               //"PLC_LED_GREEN_1" := FALSE;
               //"PLC_LED_GREEN_2" := FALSE;
               //"PLC_LED_ORANGE_1" := TRUE;
               //"PLC_LED_ORANGE_2" := FALSE;
               //"PLC_LED_GREEN_CH" := FALSE;
               //"PLC_LED_RED_1" := FALSE;
               //"PLC_LED_RED_2" := TRUE;
               //"PLC_LED_RED_CH" := TRUE;

           4:  // Statement section case S5
               // GREEN = FALSE, YELLOW = FALSE, RED = TRUE
               // PED: RED = TRUE, GREEN = FALSE

               "DB_ProcessData".crossroad_output.trafficLightEast_green := FALSE;
               "DB_ProcessData".crossroad_output.trafficLightEast_red := TRUE;
               "DB_ProcessData".crossroad_output.trafficLightEast_yellow := FALSE;

               "DB_ProcessData".crossroad_output.trafficLightNorth_green := FALSE;
               "DB_ProcessData".crossroad_output.trafficLightNorth_red := TRUE;
               "DB_ProcessData".crossroad_output.trafficLightNorth_yellow := FALSE;

               "DB_ProcessData".crossroad_output.trafficLightSouth_green := FALSE;
               "DB_ProcessData".crossroad_output.trafficLightSouth_red := TRUE;
               "DB_ProcessData".crossroad_output.trafficLightSouth_yellow := FALSE;

               "DB_ProcessData".crossroad_output.trafficLightWest_green := FALSE;
               "DB_ProcessData".crossroad_output.trafficLightWest_red := TRUE;
               "DB_ProcessData".crossroad_output.trafficLightWest_yellow := FALSE;

               "DB_ProcessData".crossroad_output.pedestrianSouth1_green := FALSE;
               "DB_ProcessData".crossroad_output.pedestrianSouth1_red := TRUE;
               "DB_ProcessData".crossroad_output.pedestrianSouth2_green := FALSE;
               "DB_ProcessData".crossroad_output.pedestrianSouth2_red := TRUE;

               "DB_ProcessData".crossroad_output.pedestrianWest1_green := FALSE;
               "DB_ProcessData".crossroad_output.pedestrianWest1_red := TRUE;
               "DB_ProcessData".crossroad_output.pedestrianWest2_green := FALSE;
               "DB_ProcessData".crossroad_output.pedestrianWest2_red := TRUE;

               //"PLC_LED_GREEN_1" := FALSE;
               //"PLC_LED_GREEN_2" := FALSE;
               //"PLC_LED_ORANGE_1" := FALSE;
               //"PLC_LED_ORANGE_2" := FALSE;
               //"PLC_LED_GREEN_CH" := FALSE;
               //"PLC_LED_RED_1" := TRUE;
               //"PLC_LED_RED_2" := TRUE;
               //"PLC_LED_RED_CH" := TRUE;

           5:  // Statement section case S6
               // GREEN = FALSE, RED = TRUE, YELLOW = FALSE   // směr 1 (East, West)
               // GREEN = FALSE, RED = TRUE, YELLOW = TRUE    // směr 2 (North, South)
               // PED: RED = TRUE, GREEN = FALSE (pokud není Crossroad_Walk_EN)

               "DB_ProcessData".crossroad_output.trafficLightEast_green := FALSE;
               "DB_ProcessData".crossroad_output.trafficLightEast_red := TRUE;
               "DB_ProcessData".crossroad_output.trafficLightEast_yellow := FALSE;

               "DB_ProcessData".crossroad_output.trafficLightNorth_green := FALSE;
               "DB_ProcessData".crossroad_output.trafficLightNorth_red := TRUE;
               "DB_ProcessData".crossroad_output.trafficLightNorth_yellow := TRUE;

               "DB_ProcessData".crossroad_output.trafficLightSouth_green := FALSE;
               "DB_ProcessData".crossroad_output.trafficLightSouth_red := TRUE;
               "DB_ProcessData".crossroad_output.trafficLightSouth_yellow := TRUE;

               "DB_ProcessData".crossroad_output.trafficLightWest_green := FALSE;
               "DB_ProcessData".crossroad_output.trafficLightWest_red := TRUE;
               "DB_ProcessData".crossroad_output.trafficLightWest_yellow := FALSE;

               "DB_ProcessData".crossroad_output.pedestrianSouth1_green := FALSE;
               "DB_ProcessData".crossroad_output.pedestrianSouth1_red := TRUE;
               "DB_ProcessData".crossroad_output.pedestrianSouth2_green := FALSE;
               "DB_ProcessData".crossroad_output.pedestrianSouth2_red := TRUE;

               "DB_ProcessData".crossroad_output.pedestrianWest1_green := FALSE;
               "DB_ProcessData".crossroad_output.pedestrianWest1_red := TRUE;
               "DB_ProcessData".crossroad_output.pedestrianWest2_green := FALSE;
               "DB_ProcessData".crossroad_output.pedestrianWest2_red := TRUE;

               //"PLC_LED_GREEN_1" := FALSE;
               //"PLC_LED_GREEN_2" := FALSE;
               //"PLC_LED_ORANGE_1" := FALSE;
               //"PLC_LED_ORANGE_2" := TRUE;
               //"PLC_LED_GREEN_CH" := FALSE;
               //"PLC_LED_RED_1" := TRUE;
               //"PLC_LED_RED_2" := TRUE;

               //"PLC_LED_GREEN_CH" := FALSE;
               //"PLC_LED_RED_CH" := TRUE;

               IF "Crossroad_Walk_EN" THEN
                   "DB_ProcessData".crossroad_output.pedestrianSouth1_green := TRUE;
                   "DB_ProcessData".crossroad_output.pedestrianSouth1_red := FALSE;
                   "DB_ProcessData".crossroad_output.pedestrianSouth2_green := TRUE;
                   "DB_ProcessData".crossroad_output.pedestrianSouth2_red := FALSE;

                   "DB_ProcessData".crossroad_output.pedestrianWest1_green := TRUE;
                   "DB_ProcessData".crossroad_output.pedestrianWest1_red := FALSE;
                   "DB_ProcessData".crossroad_output.pedestrianWest2_green := TRUE;
                   "DB_ProcessData".crossroad_output.pedestrianWest2_red := FALSE;

                   //"PLC_LED_GREEN_CH" := TRUE;
                   //"PLC_LED_RED_CH" := FALSE;
               END_IF;

           6:  // Statement section case S7
               // GREEN = FALSE, RED = TRUE, YELLOW = FALSE   // směr 1 (East, West)
               // GREEN = TRUE, RED = FALSE, YELLOW = FALSE   // směr 2 (North, South)
               // PED: RED = TRUE, GREEN = FALSE (pokud není Crossroad_Walk_EN)

               "DB_ProcessData".crossroad_output.trafficLightEast_green := FALSE;
               "DB_ProcessData".crossroad_output.trafficLightEast_red := TRUE;
               "DB_ProcessData".crossroad_output.trafficLightEast_yellow := FALSE;

               "DB_ProcessData".crossroad_output.trafficLightNorth_green := TRUE;
               "DB_ProcessData".crossroad_output.trafficLightNorth_red := FALSE;
               "DB_ProcessData".crossroad_output.trafficLightNorth_yellow := FALSE;

               "DB_ProcessData".crossroad_output.trafficLightSouth_green := TRUE;
               "DB_ProcessData".crossroad_output.trafficLightSouth_red := FALSE;
               "DB_ProcessData".crossroad_output.trafficLightSouth_yellow := FALSE;

               "DB_ProcessData".crossroad_output.trafficLightWest_green := FALSE;
               "DB_ProcessData".crossroad_output.trafficLightWest_red := TRUE;
               "DB_ProcessData".crossroad_output.trafficLightWest_yellow := FALSE;

               "DB_ProcessData".crossroad_output.pedestrianSouth1_green := FALSE;
               "DB_ProcessData".crossroad_output.pedestrianSouth1_red := TRUE;
               "DB_ProcessData".crossroad_output.pedestrianSouth2_green := FALSE;
               "DB_ProcessData".crossroad_output.pedestrianSouth2_red := TRUE;

               "DB_ProcessData".crossroad_output.pedestrianWest1_green := FALSE;
               "DB_ProcessData".crossroad_output.pedestrianWest1_red := TRUE;
               "DB_ProcessData".crossroad_output.pedestrianWest2_green := FALSE;
               "DB_ProcessData".crossroad_output.pedestrianWest2_red := TRUE;

               //"PLC_LED_GREEN_1" := FALSE;
               //"PLC_LED_GREEN_2" := TRUE;
               //"PLC_LED_ORANGE_1" := FALSE;
               //"PLC_LED_ORANGE_2" := FALSE;
               //"PLC_LED_RED_1" := TRUE;
               //"PLC_LED_RED_2" := FALSE;

               //"PLC_LED_GREEN_CH" := FALSE;
               //"PLC_LED_RED_CH" := TRUE;

               IF "Crossroad_Walk_EN" THEN
                   "DB_ProcessData".crossroad_output.pedestrianSouth1_green := TRUE;
                   "DB_ProcessData".crossroad_output.pedestrianSouth1_red := FALSE;
                   "DB_ProcessData".crossroad_output.pedestrianSouth2_green := TRUE;
                   "DB_ProcessData".crossroad_output.pedestrianSouth2_red := FALSE;

                   "DB_ProcessData".crossroad_output.pedestrianWest1_green := TRUE;
                   "DB_ProcessData".crossroad_output.pedestrianWest1_red := FALSE;
                   "DB_ProcessData".crossroad_output.pedestrianWest2_green := TRUE;
                   "DB_ProcessData".crossroad_output.pedestrianWest2_red := FALSE;

                   //"PLC_LED_GREEN_CH" := TRUE;
                   //"PLC_LED_RED_CH" := FALSE;
               END_IF;

           7:  // Statement section case S8
               // GREEN = FALSE, RED = TRUE, YELLOW = FALSE   // směr 1 (East, West)
               // GREEN = FALSE, RED = FALSE, YELLOW = TRUE   // směr 2 (North, South)
               // PED: RED = TRUE, GREEN = FALSE

               "DB_ProcessData".crossroad_output.trafficLightEast_green := FALSE;
               "DB_ProcessData".crossroad_output.trafficLightEast_red := TRUE;
               "DB_ProcessData".crossroad_output.trafficLightEast_yellow := FALSE;

               "DB_ProcessData".crossroad_output.trafficLightNorth_green := FALSE;
               "DB_ProcessData".crossroad_output.trafficLightNorth_red := FALSE;
               "DB_ProcessData".crossroad_output.trafficLightNorth_yellow := TRUE;

               "DB_ProcessData".crossroad_output.trafficLightSouth_green := FALSE;
               "DB_ProcessData".crossroad_output.trafficLightSouth_red := FALSE;
               "DB_ProcessData".crossroad_output.trafficLightSouth_yellow := TRUE;

               "DB_ProcessData".crossroad_output.trafficLightWest_green := FALSE;
               "DB_ProcessData".crossroad_output.trafficLightWest_red := TRUE;
               "DB_ProcessData".crossroad_output.trafficLightWest_yellow := FALSE;

               "DB_ProcessData".crossroad_output.pedestrianSouth1_green := FALSE;
               "DB_ProcessData".crossroad_output.pedestrianSouth1_red := TRUE;
               "DB_ProcessData".crossroad_output.pedestrianSouth2_green := FALSE;
               "DB_ProcessData".crossroad_output.pedestrianSouth2_red := TRUE;

               "DB_ProcessData".crossroad_output.pedestrianWest1_green := FALSE;
               "DB_ProcessData".crossroad_output.pedestrianWest1_red := TRUE;
               "DB_ProcessData".crossroad_output.pedestrianWest2_green := FALSE;
               "DB_ProcessData".crossroad_output.pedestrianWest2_red := TRUE;

               //"PLC_LED_GREEN_1" := FALSE;
               //"PLC_LED_GREEN_2" := FALSE;
               //"PLC_LED_ORANGE_1" := FALSE;
               //"PLC_LED_ORANGE_2" := TRUE;
               //"PLC_LED_GREEN_CH" := FALSE;
               //"PLC_LED_RED_1" := TRUE;
               //"PLC_LED_RED_2" := FALSE;
               //"PLC_LED_RED_CH" := TRUE;

           8:  // Statement section case S9
               // GREEN = FALSE, YELLOW = FALSE, RED = TRUE
               // PED: RED = TRUE, GREEN = FALSE

               "DB_ProcessData".crossroad_output.trafficLightEast_green := FALSE;
               "DB_ProcessData".crossroad_output.trafficLightEast_red := TRUE;
               "DB_ProcessData".crossroad_output.trafficLightEast_yellow := FALSE;

               "DB_ProcessData".crossroad_output.trafficLightNorth_green := FALSE;
               "DB_ProcessData".crossroad_output.trafficLightNorth_red := TRUE;
               "DB_ProcessData".crossroad_output.trafficLightNorth_yellow := FALSE;

               "DB_ProcessData".crossroad_output.trafficLightSouth_green := FALSE;
               "DB_ProcessData".crossroad_output.trafficLightSouth_red := TRUE;
               "DB_ProcessData".crossroad_output.trafficLightSouth_yellow := FALSE;

               "DB_ProcessData".crossroad_output.trafficLightWest_green := FALSE;
               "DB_ProcessData".crossroad_output.trafficLightWest_red := TRUE;
               "DB_ProcessData".crossroad_output.trafficLightWest_yellow := FALSE;

               "DB_ProcessData".crossroad_output.pedestrianSouth1_green := FALSE;
               "DB_ProcessData".crossroad_output.pedestrianSouth1_red := TRUE;
               "DB_ProcessData".crossroad_output.pedestrianSouth2_green := FALSE;
               "DB_ProcessData".crossroad_output.pedestrianSouth2_red := TRUE;

               "DB_ProcessData".crossroad_output.pedestrianWest1_green := FALSE;
               "DB_ProcessData".crossroad_output.pedestrianWest1_red := TRUE;
               "DB_ProcessData".crossroad_output.pedestrianWest2_green := FALSE;
               "DB_ProcessData".crossroad_output.pedestrianWest2_red := TRUE;

               //"PLC_LED_GREEN_1" := FALSE;
               //"PLC_LED_GREEN_2" := FALSE;
               //"PLC_LED_ORANGE_1" := FALSE;
               //"PLC_LED_ORANGE_2" := FALSE;
               //"PLC_LED_GREEN_CH" := FALSE;
               //"PLC_LED_RED_1" := TRUE;
               //"PLC_LED_RED_2" := TRUE;
               //"PLC_LED_RED_CH" := TRUE;

               "Crossroad_Walk_EN" := FALSE;

           ELSE  // Statement section ELSE
               "DB_ProcessData".crossroad_output.trafficLightEast_green := FALSE;
               "DB_ProcessData".crossroad_output.trafficLightEast_red := FALSE;
               "DB_ProcessData".crossroad_output.trafficLightEast_yellow := FALSE;

               "DB_ProcessData".crossroad_output.trafficLightNorth_green := FALSE;
               "DB_ProcessData".crossroad_output.trafficLightNorth_red := FALSE;
               "DB_ProcessData".crossroad_output.trafficLightNorth_yellow := FALSE;

               "DB_ProcessData".crossroad_output.trafficLightSouth_green := FALSE;
               "DB_ProcessData".crossroad_output.trafficLightSouth_red := FALSE;
               "DB_ProcessData".crossroad_output.trafficLightSouth_yellow := FALSE;

               "DB_ProcessData".crossroad_output.trafficLightWest_green := FALSE;
               "DB_ProcessData".crossroad_output.trafficLightWest_red := FALSE;
               "DB_ProcessData".crossroad_output.trafficLightWest_yellow := FALSE;

               "DB_ProcessData".crossroad_output.pedestrianSouth1_green := FALSE;
               "DB_ProcessData".crossroad_output.pedestrianSouth1_red := FALSE;
               "DB_ProcessData".crossroad_output.pedestrianSouth2_green := FALSE;
               "DB_ProcessData".crossroad_output.pedestrianSouth2_red := FALSE;

               "DB_ProcessData".crossroad_output.pedestrianWest1_green := FALSE;
               "DB_ProcessData".crossroad_output.pedestrianWest1_red := FALSE;
               "DB_ProcessData".crossroad_output.pedestrianWest2_green := FALSE;
               "DB_ProcessData".crossroad_output.pedestrianWest2_red := FALSE;

               //"PLC_LED_GREEN_1" := FALSE;
               //"PLC_LED_GREEN_2" := FALSE;
               //"PLC_LED_ORANGE_1" := FALSE;
               //"PLC_LED_ORANGE_2" := FALSE;
               //"PLC_LED_RED_1" := FALSE;
               //"PLC_LED_RED_2" := FALSE;
               //"PLC_LED_GREEN_CH" := FALSE;
               //"PLC_LED_RED_CH" := FALSE;

               "Crossroad_Walk_EN" := FALSE;
       END_CASE;
   END_IF;
END_REGION

REGION Network 6 (SCL): Pedestrians bnts
   IF "DB_ProcessData".crossroad_input.btnSouthCrosswalk1 OR "DB_ProcessData".crossroad_input.btnSouthCrosswalk2 OR "DB_ProcessData".crossroad_input.btnWestCrosswalk1 OR "DB_ProcessData".crossroad_input.btnWestCrosswalk2 THEN
       "Crossroad_Walk_EN" := TRUE;
   END_IF;
END_REGION
END_FUNCTION

// folder: Crosswalk

FUNCTION "Crosswalk_MAIN" : Void   // FC1, LAD
{ S7_Optimized_Access := 'TRUE' }
VERSION : 0.1
BEGIN

REGION Network 1: Control
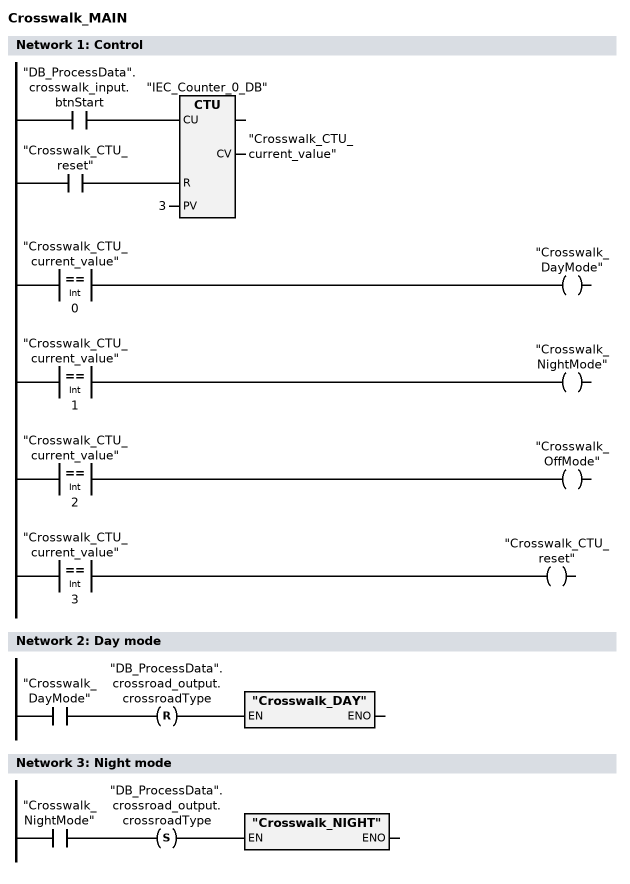
   "IEC_Counter_0_DB".CTU(CU := "DB_ProcessData".crosswalk_input.btnStart,
                          R := "Crosswalk_CTU_reset",
                          PV := 3,
                          CV => "Crosswalk_CTU_current_value");
   "Crosswalk_DayMode" := "Crosswalk_CTU_current_value" = 0;
   "Crosswalk_NightMode" := "Crosswalk_CTU_current_value" = 1;
   "Crosswalk_OffMode" := "Crosswalk_CTU_current_value" = 2;
   "Crosswalk_CTU_reset" := "Crosswalk_CTU_current_value" = 3;
END_REGION

REGION Network 2: Day mode
   RUNG wire#powerrail
      Contact( "Crosswalk_DayMode" )
      R_Coil( "DB_ProcessData".crossroad_output.crossroadType )
      "Crosswalk_DAY"()
   END_RUNG
   // the same network as SCL:
   IF "Crosswalk_DayMode" THEN
       "DB_ProcessData".crossroad_output.crossroadType := FALSE;
       "Crosswalk_DAY"();
   END_IF;
END_REGION

REGION Network 3: Night mode
   RUNG wire#powerrail
      Contact( "Crosswalk_NightMode" )
      S_Coil( "DB_ProcessData".crossroad_output.crossroadType )
      "Crosswalk_NIGHT"()
   END_RUNG
   // the same network as SCL:
   IF "Crosswalk_NightMode" THEN
       "DB_ProcessData".crossroad_output.crossroadType := TRUE;
       "Crosswalk_NIGHT"();
   END_IF;
END_REGION

REGION Network 4 (SCL): Off mode
   IF "Crosswalk_OffMode" = TRUE THEN
       "DB_ProcessData".crosswalk_output.pedestrianLightGreen1 := FALSE;
       "DB_ProcessData".crosswalk_output.pedestrianLightGreen2 := FALSE;
       "DB_ProcessData".crosswalk_output.pedestrianLightRed1 := FALSE;
       "DB_ProcessData".crosswalk_output.pedestrianLightRed2 := FALSE;
       "DB_ProcessData".crosswalk_output.trafficLightGreen1 := FALSE;
       "DB_ProcessData".crosswalk_output.trafficLightGreen2 := FALSE;
       "DB_ProcessData".crosswalk_output.trafficLightsRed1 := FALSE;
       "DB_ProcessData".crosswalk_output.trafficLightsRed2 := FALSE;
       "DB_ProcessData".crosswalk_output.trafficLightsYellow1 := FALSE;
       "DB_ProcessData".crosswalk_output.trafficLightsYellow2 := FALSE;
   END_IF;
END_REGION
END_FUNCTION

FUNCTION "Crosswalk_DAY" : Void   // FC2, LAD
{ S7_Optimized_Access := 'TRUE' }
VERSION : 0.1
   VAR_TEMP   // added for the SCL form of the ladder/FBD networks
      _w1 : Bool;
   END_VAR
BEGIN

REGION Network 1: Green
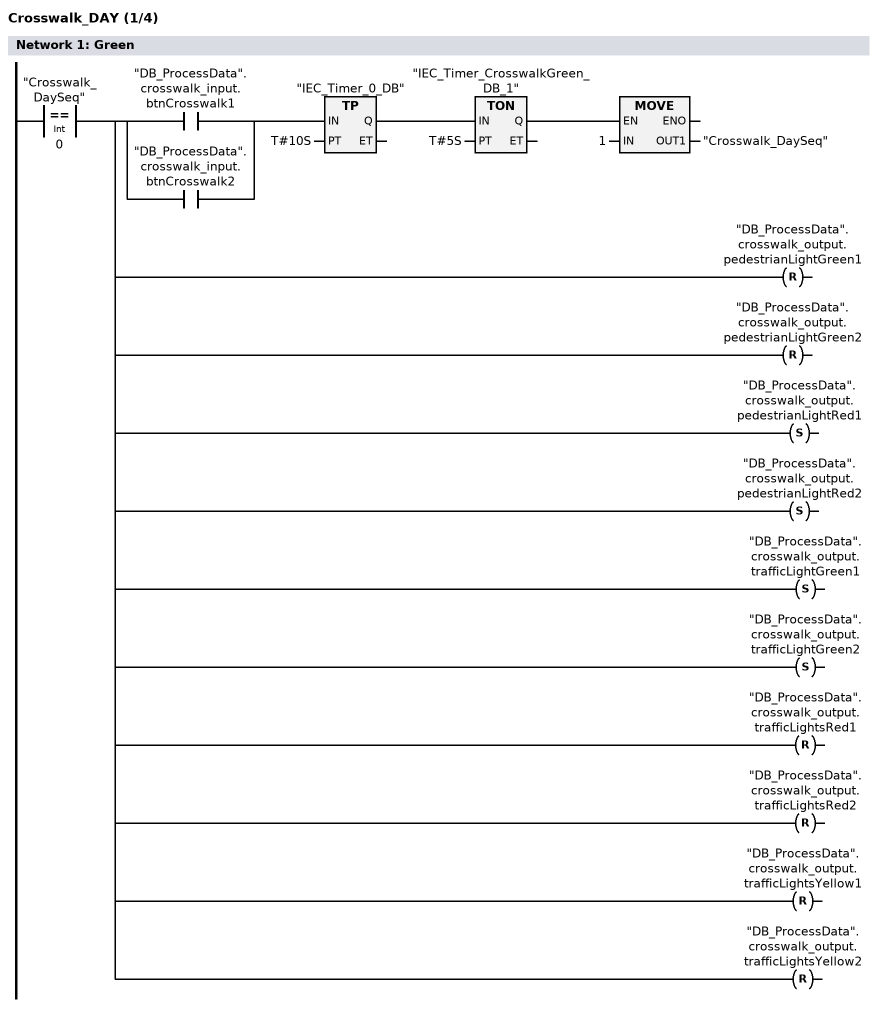
   #_w1 := "Crosswalk_DaySeq" = 0;
   "IEC_Timer_0_DB".TP(IN := #_w1 AND ("DB_ProcessData".crosswalk_input.btnCrosswalk1 OR "DB_ProcessData".crosswalk_input.btnCrosswalk2),
                       PT := T#10S);
   "IEC_Timer_CrosswalkGreen_DB_1".TON(IN := "IEC_Timer_0_DB".Q, PT := T#5S);
   IF "IEC_Timer_CrosswalkGreen_DB_1".Q THEN "Crosswalk_DaySeq" := 1; END_IF;
   IF #_w1 THEN
       "DB_ProcessData".crosswalk_output.pedestrianLightGreen1 := FALSE;
       "DB_ProcessData".crosswalk_output.pedestrianLightGreen2 := FALSE;
       "DB_ProcessData".crosswalk_output.pedestrianLightRed1 := TRUE;
       "DB_ProcessData".crosswalk_output.pedestrianLightRed2 := TRUE;
       "DB_ProcessData".crosswalk_output.trafficLightGreen1 := TRUE;
       "DB_ProcessData".crosswalk_output.trafficLightGreen2 := TRUE;
       "DB_ProcessData".crosswalk_output.trafficLightsRed1 := FALSE;
       "DB_ProcessData".crosswalk_output.trafficLightsRed2 := FALSE;
       "DB_ProcessData".crosswalk_output.trafficLightsYellow1 := FALSE;
       "DB_ProcessData".crosswalk_output.trafficLightsYellow2 := FALSE;
   END_IF;
END_REGION

REGION Network 2: Yellow1
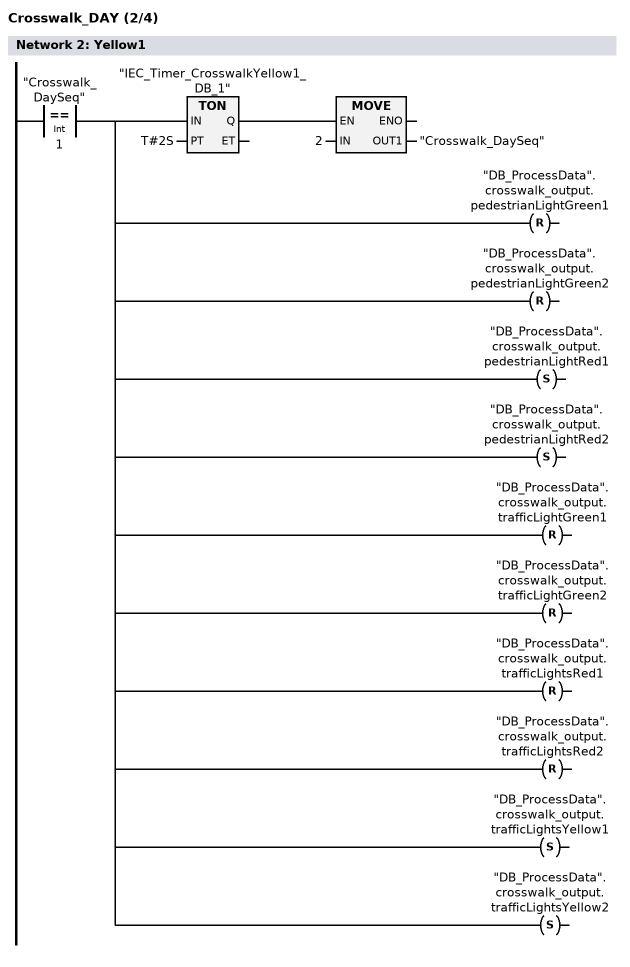
   #_w1 := "Crosswalk_DaySeq" = 1;
   "IEC_Timer_CrosswalkYellow1_DB_1".TON(IN := #_w1, PT := T#2S);
   IF "IEC_Timer_CrosswalkYellow1_DB_1".Q THEN "Crosswalk_DaySeq" := 2; END_IF;
   IF #_w1 THEN
       "DB_ProcessData".crosswalk_output.pedestrianLightGreen1 := FALSE;
       "DB_ProcessData".crosswalk_output.pedestrianLightGreen2 := FALSE;
       "DB_ProcessData".crosswalk_output.pedestrianLightRed1 := TRUE;
       "DB_ProcessData".crosswalk_output.pedestrianLightRed2 := TRUE;
       "DB_ProcessData".crosswalk_output.trafficLightGreen1 := FALSE;
       "DB_ProcessData".crosswalk_output.trafficLightGreen2 := FALSE;
       "DB_ProcessData".crosswalk_output.trafficLightsRed1 := FALSE;
       "DB_ProcessData".crosswalk_output.trafficLightsRed2 := FALSE;
       "DB_ProcessData".crosswalk_output.trafficLightsYellow1 := TRUE;
       "DB_ProcessData".crosswalk_output.trafficLightsYellow2 := TRUE;
   END_IF;
END_REGION

REGION Network 3: Red
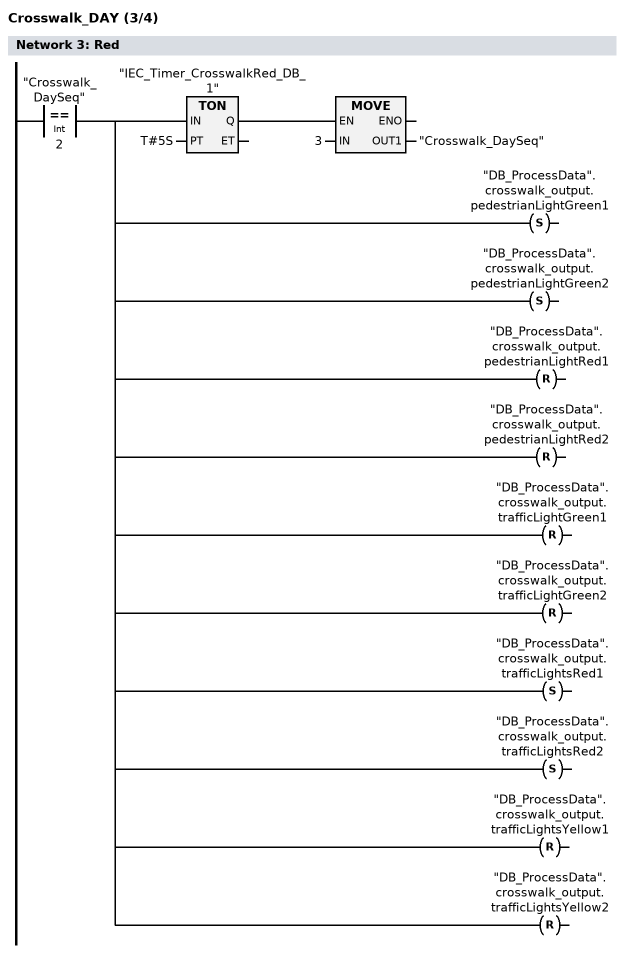
   #_w1 := "Crosswalk_DaySeq" = 2;
   "IEC_Timer_CrosswalkRed_DB_1".TON(IN := #_w1, PT := T#5S);
   IF "IEC_Timer_CrosswalkRed_DB_1".Q THEN "Crosswalk_DaySeq" := 3; END_IF;
   IF #_w1 THEN
       "DB_ProcessData".crosswalk_output.pedestrianLightGreen1 := TRUE;
       "DB_ProcessData".crosswalk_output.pedestrianLightGreen2 := TRUE;
       "DB_ProcessData".crosswalk_output.pedestrianLightRed1 := FALSE;
       "DB_ProcessData".crosswalk_output.pedestrianLightRed2 := FALSE;
       "DB_ProcessData".crosswalk_output.trafficLightGreen1 := FALSE;
       "DB_ProcessData".crosswalk_output.trafficLightGreen2 := FALSE;
       "DB_ProcessData".crosswalk_output.trafficLightsRed1 := TRUE;
       "DB_ProcessData".crosswalk_output.trafficLightsRed2 := TRUE;
       "DB_ProcessData".crosswalk_output.trafficLightsYellow1 := FALSE;
       "DB_ProcessData".crosswalk_output.trafficLightsYellow2 := FALSE;
   END_IF;
END_REGION

REGION Network 4: Yellow2
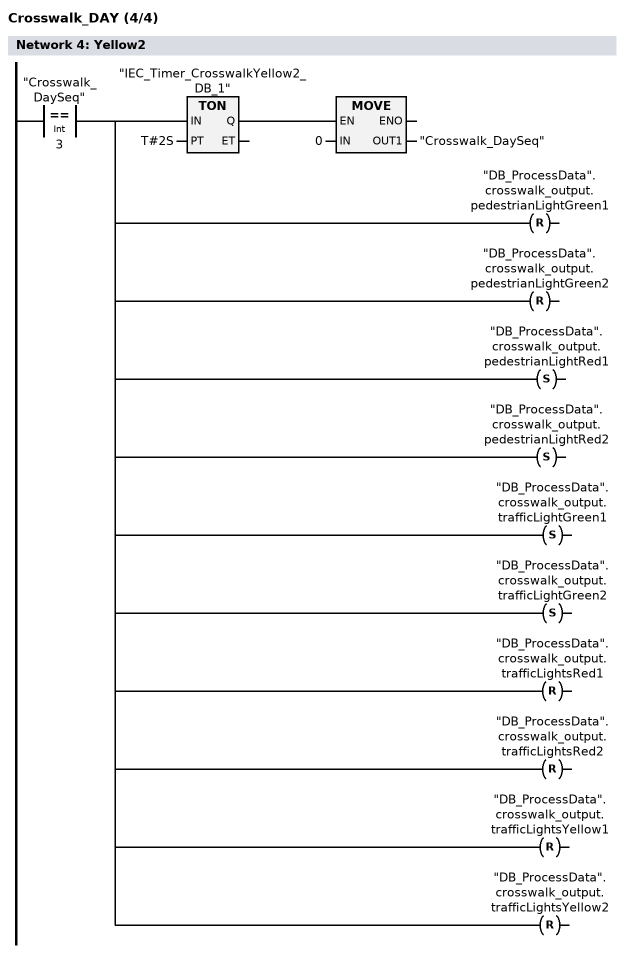
   #_w1 := "Crosswalk_DaySeq" = 3;
   "IEC_Timer_CrosswalkYellow2_DB_1".TON(IN := #_w1, PT := T#2S);
   IF "IEC_Timer_CrosswalkYellow2_DB_1".Q THEN "Crosswalk_DaySeq" := 0; END_IF;
   IF #_w1 THEN
       "DB_ProcessData".crosswalk_output.pedestrianLightGreen1 := FALSE;
       "DB_ProcessData".crosswalk_output.pedestrianLightGreen2 := FALSE;
       "DB_ProcessData".crosswalk_output.pedestrianLightRed1 := TRUE;
       "DB_ProcessData".crosswalk_output.pedestrianLightRed2 := TRUE;
       "DB_ProcessData".crosswalk_output.trafficLightGreen1 := TRUE;
       "DB_ProcessData".crosswalk_output.trafficLightGreen2 := TRUE;
       "DB_ProcessData".crosswalk_output.trafficLightsRed1 := FALSE;
       "DB_ProcessData".crosswalk_output.trafficLightsRed2 := FALSE;
       "DB_ProcessData".crosswalk_output.trafficLightsYellow1 := FALSE;
       "DB_ProcessData".crosswalk_output.trafficLightsYellow2 := FALSE;
   END_IF;
END_REGION
END_FUNCTION

FUNCTION "Crosswalk_NIGHT" : Void   // FC3, LAD
{ S7_Optimized_Access := 'TRUE' }
VERSION : 0.1
   VAR_TEMP   // added for the SCL form of the ladder/FBD networks
      _w1 : Bool;
   END_VAR
BEGIN

REGION Network 1: On
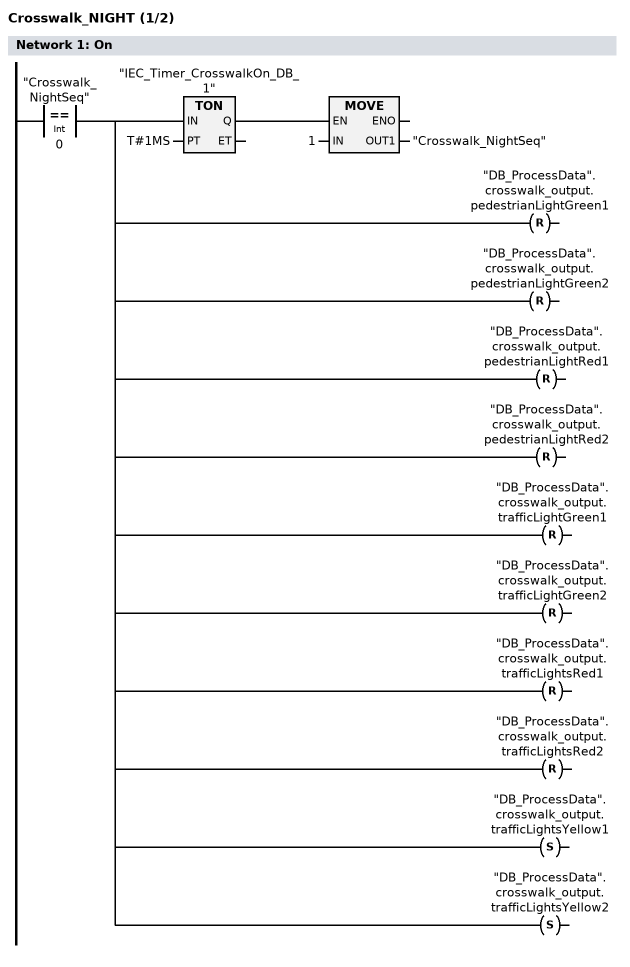
   #_w1 := "Crosswalk_NightSeq" = 0;
   "IEC_Timer_CrosswalkOn_DB_1".TON(IN := #_w1, PT := T#1MS);
   IF "IEC_Timer_CrosswalkOn_DB_1".Q THEN "Crosswalk_NightSeq" := 1; END_IF;
   IF #_w1 THEN
       "DB_ProcessData".crosswalk_output.pedestrianLightGreen1 := FALSE;
       "DB_ProcessData".crosswalk_output.pedestrianLightGreen2 := FALSE;
       "DB_ProcessData".crosswalk_output.pedestrianLightRed1 := FALSE;
       "DB_ProcessData".crosswalk_output.pedestrianLightRed2 := FALSE;
       "DB_ProcessData".crosswalk_output.trafficLightGreen1 := FALSE;
       "DB_ProcessData".crosswalk_output.trafficLightGreen2 := FALSE;
       "DB_ProcessData".crosswalk_output.trafficLightsRed1 := FALSE;
       "DB_ProcessData".crosswalk_output.trafficLightsRed2 := FALSE;
       "DB_ProcessData".crosswalk_output.trafficLightsYellow1 := TRUE;
       "DB_ProcessData".crosswalk_output.trafficLightsYellow2 := TRUE;
   END_IF;
END_REGION

REGION Network 2: Off
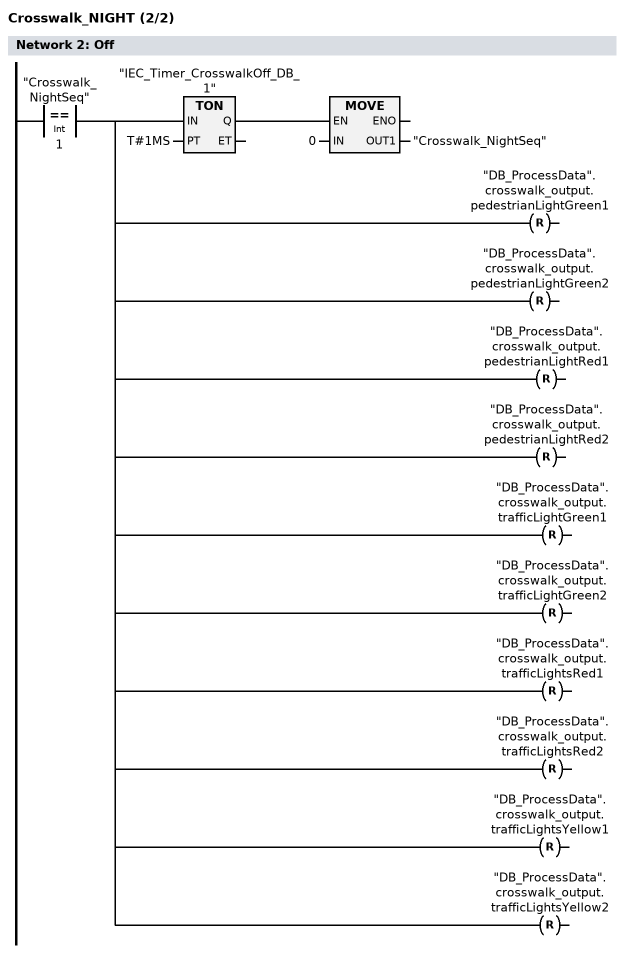
   #_w1 := "Crosswalk_NightSeq" = 1;
   "IEC_Timer_CrosswalkOff_DB_1".TON(IN := #_w1, PT := T#1MS);
   IF "IEC_Timer_CrosswalkOff_DB_1".Q THEN "Crosswalk_NightSeq" := 0; END_IF;
   IF #_w1 THEN
       "DB_ProcessData".crosswalk_output.pedestrianLightGreen1 := FALSE;
       "DB_ProcessData".crosswalk_output.pedestrianLightGreen2 := FALSE;
       "DB_ProcessData".crosswalk_output.pedestrianLightRed1 := FALSE;
       "DB_ProcessData".crosswalk_output.pedestrianLightRed2 := FALSE;
       "DB_ProcessData".crosswalk_output.trafficLightGreen1 := FALSE;
       "DB_ProcessData".crosswalk_output.trafficLightGreen2 := FALSE;
       "DB_ProcessData".crosswalk_output.trafficLightsRed1 := FALSE;
       "DB_ProcessData".crosswalk_output.trafficLightsRed2 := FALSE;
       "DB_ProcessData".crosswalk_output.trafficLightsYellow1 := FALSE;
       "DB_ProcessData".crosswalk_output.trafficLightsYellow2 := FALSE;
   END_IF;
END_REGION
END_FUNCTION

// folder: LMQTT

FUNCTION_BLOCK "LMQTT_Client"   // FB11, SCL
TITLE = LMQTT_Client
{ S7_Optimized_Access := 'TRUE' }
AUTHOR : Siemens Industry Online Support
FAMILY : LMQTT
VERSION : 4.0
// This block allows to connect to an MQTT Broker and publish data or receive data via a subscription.
   VAR_INPUT
      enable : Bool;   // Set TRUE, to establish a connection - set to FALSE to disconnect
      publish : Bool;   // Rising Edge: Sends a message
      subscribe : Bool;   // Rising Edge: Subscribes to a topic
      unsubscribe : Bool;   // Rising Edge: Unsubscribes to a topic
      qos : USInt;   // Quality of Service for publish/subscribe requests and last will. Subscribe only allows QoS 0 and 1
      retain : Bool;   // TRUE: Published Message will be set to retain on MQTT broker
      publishMsgLen : UDInt := 0;   // Valid number of elements in publish message data Array
      willMsgLen : UInt := 0;   // Valid number of elements in Will Message Data Array. Max 65535 Byte allowed by MQTT Spec.
      timeOut : Time := T#5s;   // Sets the time out value for every request (publish/subscribe/unsubscribe/ping)
   END_VAR
   VAR_OUTPUT
      valid : Bool;   // TRUE: Valid set of output values available at the FB
      done : Bool;   // TRUE: If last Request was successfull
      busy : Bool;   // TRUE: FB is not finished and new output values can be expected
      error : Bool;   // TRUE: An error occurred during the execution of the FB
      status : Word := 16#7000;   // 16#0000 - 16#7FFF: Status of the FB, 16#8000 - 16#FFFF: Error identification
      diagnostics : "typeDiagnostics";   // Diagnostics information of FB
      receivedMsgStatus : USInt;   // 0: No new Message, 1: New valid Message received and available at InOut area, 2: New message, but data is invalid (wrong message len or message could not be copied to InOut received topic or received message)
      receivedMsgDataLen : UDInt;   // Amount of Bytes received in receivedMessage INOUT area
   END_VAR
   VAR_IN_OUT
      connParam : "LMQTT_typeConnParam";   // Connection parameters
      clientIdentifier : WString;   // Client identifier
      username : WString;   // Username to connect
      password : WString;   // Password to connect
      willtopic : WString;   // Topic where the last will message is sent
      willMsgPayload : Array[*] of Byte;   // Last will message Data - valid bytes in this array must be written in input 'willMsgLen'
      mqttTopic : WString;   // Mqtt Topic to Publish / Subscribe / Unsubscribe
      publishMsgPayload : Array[*] of Byte;   // Message Data to Publish - valid bytes in this array must be written in input 'publishMsgLen'
      receivedTopic : WString;   // Mqtt Topic of received message
      receivedMsgPayload : Array[*] of Byte;   // Mqtt message data that was received - valid bytes in this array indicated by 'receivedMsgDataLen' output
   END_VAR
   VAR
      statEnableOld : Bool;   // Old value of 'enable' input for edge detection
      statValid : Bool;   // Static value for output 'valid'
      statBusy : Bool;   // Static value for output 'busy'
      statError : Bool;   // Static value for output 'error'
      statErrorUserCleared : Bool;   // Error occurred that can only be solved by user; rising edge at enable input necessary
      statErrorAutoCleared : Bool;   // Error occurred that can be acknowledged by FB
      statStatus : Word := 16#7000;   // Static value for output 'status'
      statDone : Bool;   // Static value for output 'done'
      statRcvMsgStatus : USInt;   // Static value for output 'receivedMsgStatus'
      statRcvMsgDataLen : UDInt;   // Static value for output 'receivedMsgDataLen'
      statSubfunctionStatus : Word;   // Status or return value of called FBs, FCs and system blocks
      statFBErrorState : DInt;   // State in the state machine of the block where the error occurred
      statFBState : DInt := 0;   // State in the state machine of the FB
      statMqttConnectState : DInt := 0;   // State in the state machine of the MQTT Connection
      statMqttCommandState : DInt := 0;   // State in the state machine of the MQTT Commands when MQTT is connected
      statDisablingCompleted : Bool;   // TRUE: Disabling has been completed
      statEmptyDiagnostics : "typeDiagnostics";   // Empty diagnostics information (for initialization purposes only)
      statConnParam : Struct   // Connection parameters
         isQDN : Bool;   // QDN is used instead of IP address
         paramQDN : TCON_QDN_SEC;   // Parameter to assign QDN information
         paramIP : TCON_IP_V4_SEC;   // Parameter to assign IP information
      END_STRUCT;
      instTsendC : TSEND_C;   // Tsend Instance
      instTrcv : TRCV;   // Trcv Instance
      statSendBuffer : Array[0..#MAX_BUFFER_LEN_SEND] of Byte;   // Send buffer to send Data via TSend
      statRcvBuffer : Array[0..#MAX_BUFFER_LEN_RCV] of Byte;   // Receive buffer to receive Data via Trcv
      statPublishOld : Bool;   // Old value of 'publish' input for edge detection
      statSubscribeOld : Bool;   // Old value of 'subscribe' input for edge detection
      statUnsubscribeOld : Bool;   // Old value of 'unsubscribe' input for edge detection
      statTsendcReq : Bool;   // Static value to set send request
      statTsendcEnable : Bool;   // Static value to set tsend to enabled
      statTsendcLen : UDInt;   // Static value to len of tsend block
      statEnableTimerCommandWatchdog : Bool;   // Static value to start the command timer timeout
      instTimerCommandWatchdog : IEC_TIMER;   // Instance of the Timer for commands
      statEnableMqttKeepAliveTimer : Bool;   // Static value to enable the Mqtt keepalive timer
      statMqttKeepAliveUsed : Bool;   // Static value to show if keepalive is used or deactivated
      statMqttKeepAliveTime : Time;   // Static value to store the keepalive Time interval
      instMqttKeepAliveTimer : IEC_TIMER;   // Instance of the Timer for Mqtt keepalive
      statSendBufferPos : UInt;   // Static value to store the buffer position of the Tsend data area
      statPaketHeaderEncodeDone : Bool;   // Static value to show if a paket header was already encoded
      statSendPaketTotalRemLen : UDInt;   // Static value to store total paket length in bytes
      statEncodedRemPaketLenAsByte : Byte;   // Static value to store remaining length encoded as byte during calculation
      statUsernameLenUtf8Encoded : UInt;   // Static value to store total length of the username in utf8
      statPasswordLenUtf8Encoded : UInt;   // Static value to store total length of the password in utf8
      statWillTopicLenUtf8Encoded : UInt;   // Static value to store total length of the will topic in utf8
      statClientIdLenUtf8Encoded : UInt;   // Static value to store total length of the client id in utf8
      statWillQos : USInt;   // Static value to store the qos information of the will message
      statWillRetain : Bool;   // Static value to store the retain information of the will message
      statWillMessageCnt : UInt;   // Static value to store the amount of valid bytes in will message array
      statClientIdPos : DInt;   // Static value to store client id position during encoding
      statClientIdEncodeState : DInt;   // Static value to store the state during encoding
      statWillMessagePos : DInt;   // Static value to store will message position during encoding
      statWillMessageEncodeState : DInt;   // Static value to store the state during encoding
      statWillTopicPos : DInt;   // Static value to store will topic position during encoding
      statWillTopicEncodeState : DInt;   // Static value to store the state during encoding
      statUserNamePos : DInt;   // Static value to store user name position during encoding
      statUserNameEncodeState : DInt;   // Static value to store the state during encoding
      statPasswordPos : DInt;   // Static value to store password position during encoding
      statPasswordEncodeState : DInt;   // Static value to store the state during encoding
      statPaketId : UInt;   // Static value for the PaketId of each sent paket
      statPublishTopicLenUtf8Encoded : UInt;   // Static value to store total length of the publish topic in utf8
      statPublishQos : USInt;   // Static value to store the qos information of the publish message
      statPublishMessageCnt : UDInt;   // Static value to store the amount of valid bytes in publish message array
      statPublishTopicEncodeState : DInt;   // Static value to store the state during encoding
      statPublishTopicPos : DInt;   // Static value to store publish topic position during encoding
      statPaketIdEncoded : Bool;   // Static value to store if the paket id was encoded
      statPublishEncodeMessageState : DInt;   // Static value to store the state during encoding
      statPublishMessagePos : DInt;   // Static value to store publish message position during encoding
      statSubscribeQos : USInt;   // Static value to store the qos information of the subscribe message
      statSubscribeQosEncoded : Bool;   // Static value to store if the qos was encoded
      statSubscribeTopicPos : DInt;   // Static value to store subscribe topic position during encoding
      statSubscribeTopicEncodeState : DInt;   // Static value to store the state during encoding
      statSubscribeTopicLenUtf8Encoded : UInt;   // Static value to store total length of the subscribe topic in utf8
      statUnsubscribeTopicPos : DInt;   // Static value to store unsubscribe topic position during encoding
      statUnsubscribeTopicEncodeState : DInt;   // Static value to store the state during encoding
      statUnsubscribeTopicLenUtf8Encoded : UInt;   // Static value to store total length of the unsubscribe topic in utf8
      statRcvMsgQoS : UInt;   // Static value to store the qos information of the received message
      statRcvMsgTotalLen : UDInt;   // Static value to store the total len of the received message
      statRcvMsgTopicLen : UInt;   // Static value to store the total len of the received message topic
      statRcvMsgPayloadLen : UDInt;   // Static value to store the total len of the received message payload
      statRcvMsgPaketId : Word;   // Static value to store the paket id of the received message
      statRcvMsgTopicPos : DInt;   // Static value to store received message topic position during decoding
      statRcvMsgPayloadPos : DInt;   // Static value to store received message payload position during decoding
      statRcvMsgDecodeState : DInt;   // State in the state machine of the Rcv decoding
      statRcvMsgInternalStatus : USInt;   // Static value to store the internal status in case of topic or payload overflow
      statMqttPubRecRcv : USInt;   // Temporary value to store Publish Received of mqtt broker
      statSendPubAckMsg : Bool;   // Static value to signal if publish acknowledge message must be sent
      statPubRecReady : Bool;
      statCommandInputOld : Bool;
      statCommandInputBackup : Byte;
   END_VAR
   VAR_TEMP
      tempEnable : Bool;   // Temporary value for input 'enable'
      tempSubscribe : Bool;   // Temporary value for input 'subscribe'
      tempPublish : Bool;   // Temporary value for input 'publish'
      tempUnsubscribe : Bool;   // Temporary value for input 'unsubscribe'
      tempTsendcDone : Bool;   // Temporary value for instance of TsendC
      tempTsendcBusy : Bool;   // Temporary value for instance of TsendC
      tempTsendcError : Bool;   // Temporary value for instance of TsendC
      tempTsendcStatus : Word;   // Temporary value for instance of TsendC
      tempTrcvNdr : Bool;   // Temporary value for instance of Trcv
      tempTrcvBusy : Bool;   // Temporary value for instance of Trcv
      tempTrcvError : Bool;   // Temporary value for instance of Trcv
      tempTrcvStatus : Word;   // Temporary value for instance of Trcv
      tempTrcvRcvdLen : UDInt;   // Temporary value for instance of Trcv
      tempTrcvBufferPos : DInt;   // Temporary value for buffer position in trcv data array
      tempUserFlag : Bool;   // Temporary value to indicate if username is set
      tempPasswordFlag : Bool;   // Temporary value to indicate if passwordis set
      tempWillFlag : Bool;   // Temporary value to indicate if last will is set
      tempWillQoS1 : Bool;   // Temporary value to indicate if lastwill uses qos 1
      tempWillQoS2 : Bool;   // Temporary value to indicate if lastwill uses qos 2
      tempMaxWillMsgLen : DInt;   // Temporary value to store max will msg len
      tempLowerWillMsgArrayBoundary : DInt;   // Temporary value to store will msg data array lower bound from inout
      tempLoopCounter : DInt;   // Temporary value for several For loops
      tempBytesUsedUtf8 : USInt;   // Temporary value to store bytes used by a single character
      tempErrorConvertUtf8 : Bool;   // Temporary value to store if an error occured while converting character to utf8
      tempStatusConvertUtf8 : Word;   // Temporary value to store status code while converting character to utf8
      tempConvertedUtf8 : DWord;   // Temporary value to store the converted character in utf-8 format
      tempWordForSliceAddress : Word;   // Temporary value for several slice accesses
      tempCommandInput : Byte;   // Temporary value to set wether the command was publish subscribe or unsubscribe
      tempRcvMsgTypeCase : Byte;   // Temporary value to store which message type was received
      tempMaxPublishDataArrayLen : DInt;   // Temporary value to store the total length of the publish msg data array at inout
      tempMqttConnAckRcvStatus : USInt;   // Temporary value to store state of connection acknowledgement from broker
      tempMqttPingRspRcv : USInt;   // Temporary value to store PingResponse from broker
      tempMqttPubAckRcv : USInt;   // Temporary value to store Publish acknowledgement of mqtt broker
      tempMqttPubCompRcv : USInt;   // Temporary value to store Publish Completed of mqtt broker
      tempMqttSubAckRcv : USInt;   // Temporary value to store Subscribe acknowledgement of mqtt broker
      tempMqttUnSubAckRcv : USInt;   // Temporary value to store Unsubscribe acknowledgement of mqtt broker
      tempLowerBoundPublishDataArray : DInt;   // Temporary value to store lower bound of the publish data array
      tempMultiplierToDecode : UDInt;   // Temporary value to store the multiplier while paket decoding algorithm
      tempReceivedTopicStringMaxLen : DInt;   // Temporary value to store the max string len of the received topic
      tempReceivedMsgDataArrayTotalLen : DInt;   // Temporary value to store the total len of the received data msg array at inout
      tempUpperBoundRcvMsgDataArray : DInt;   // Temporary value to store the upper bound of the msg payload array
      tempFirstChar : Int;   // First character of broker address as numeric value
   END_VAR
   VAR CONSTANT
      FB_STATE_NO_PROCESSING : DInt := 0;   // FB state: No processing
      FB_STATE_VALIDATE_INPUT : DInt := 10;   // FB state: Enabling - Validation of Inputs
      FB_STATE_TCP_CONNECTING : DInt := 20;   // FB state: Processing - TCP Connection establishing
      FB_STATE_OPERATING_MONITOR_TCP : DInt := 30;   // FB state: Processing - TCP Established, MQTT connection in progress
      FB_STATE_TCP_RECONNECTING : DInt := 40;   // FB state: Processing - TCP Connection must be re-established
      FB_STATE_DISABLING : DInt := 90;   // FB state: Disabling
      MQTT_CONNECT_STATE_NO_PROCESSING : DInt := 0;   // MQTT state: No processing
      MQTT_CONNECT_STATE_BUILD_PAKET : DInt := 100;   // MQTT state: Processing - build connect paket
      MQTT_CONNECT_STATE_SEND_PAKET_WAIT_FOR_CONNACK : DInt := 200;   // MQTT state: Processing - send connect paket
      MQTT_CONNECT_STATE_CONNECTED : DInt := 300;   // MQTT state: Processing - Connected to MQTT Broker
      MQTT_CONNECT_STATE_DISCONNECTED : DInt := 400;   // MQTT state: Processing - Disconnected to MQTT Broker
      MQTT_COMMAND_STATE_NO_PROCESSING : DInt := 0;   // MQTT Command state: No processing
      MQTT_COMMAND_STATE_BUILD_PUBLISH : DInt := 1;   // MQTT Command state: Build Publish paket
      MQTT_COMMAND_STATE_SEND_PUBLISH : DInt := 1000;   // MQTT Command state: Send Publish paket
      MQTT_COMMAND_STATE_BUILD_SUBSCRIBE : DInt := 2;   // MQTT Command state: Build Subscribe paket
      MQTT_COMMAND_STATE_SEND_SUBSCRIBE : DInt := 2000;   // MQTT Command state: Send Subscribe paket
      MQTT_COMMAND_STATE_BUILD_UNSUBSCRIBE : DInt := 4;   // MQTT Command state: Build Unsubscribe paket
      MQTT_COMMAND_STATE_SEND_UNSUBSCRIBE : DInt := 3000;   // MQTT Command state: Send Unsubscribe paket
      MQTT_COMMAND_STATE_SEND_PING : DInt := 8000;   // MQTT Command state: Send Ping paket
      MQTT_COMMAND_STATE_PING_RESP : DInt := 9000;   // MQTT Command state: Receive Ping paket
      STATUS_JOB_EXECUTED : Word := 16#0000;   // The last job was successfully executed
      STATUS_NO_CALL : Word := 16#7000;   // No job being currently processed
      STATUS_FIRST_CALL : Word := 16#7001;   // First call after incoming new job (rising edge 'enable')
      STATUS_SUBSEQUENT_CALL : Word := 16#7002;   // Subsequent call during active processing without further details
      STATUS_MQTT_CONNECTING : Word := 16#7003;   // Currently connecting to MQTT Broker
      STATUS_MQTT_CONNECTED : Word := 16#7004;   // Connected to MQTT Broker
      STATUS_MQTT_PING : Word := 16#7005;   // Processing Ping to Broker
      STATUS_MQTT_PUBLISH : Word := 16#7006;   // Processing Publish to Broker
      STATUS_MQTT_SUBSCRIBE : Word := 16#7008;   // Processing Subscribe to Broker
      STATUS_MQTT_UNSUBSCRIBE : Word := 16#7010;   // Processing Unsubscribe to Broker
      ERR_UNDEFINED_STATE : Word := 16#8600;   // Error due to an undefined state in state machine
      ERR_TCP_RECONNECTING : Word := 16#9000;   // Error, lost connection to mqtt broker, reconnect ongoing
      ERR_CLIENT_ID_NULL : Word := 16#8200;   // Error due to an incorrect client id at input
      ERR_BROKER_INVALID : Word := 16#8201;   // Error: Parameter "broker" is invalid
      ERR_CNT_EXCEEDS_ARRAY_DIMENSION : Word := 16#8210;   // Error due to an incorrect assignment of publish msg len or will msg len
      ERR_KEEPALIVE_INVALID : Word := 16#8220;   // Error due to an incorrect assignment of keepalive input
      ERR_QOS_INVALID : Word := 16#8230;   // Error due to an incorrect assignment of qos input
      ERR_TCON_FAILED : Word := 16#8601;   // Error while trying to connect to mqtt broker with tcon
      ERR_TCON_TIMEOUT : Word := 16#8620;   // Error due to time out while trying to connect to broker
      ERR_MQTT_REM_LEN_INVALID : Word := 16#8700;   // Error due to receiving an invalid mqtt paket
      ERR_MQTT_MALFORMED_QOS_RECEIVED : Word := 16#8710;   // Error due to receiving an invalid mqtt paket
      ERR_MQTT_CONNACK_INVALID_SESSION_FLAG : Word := 16#8720;   // Error due to receiving an invalid mqtt paket
      ERR_MQTT_CONNACK_RETURN_CODE_INVALID : Word := 16#8730;   // Error due to receiving an invalid mqtt paket - see subfunction status for more information
      ERR_MQTT_PAKET_ID_INVALID : Word := 16#8740;   // Error due to receiving an invalid mqtt paket id
      ERR_MQTT_SUBACK_FAILURE : Word := 16#8750;   // Error because of failing to create a subscription
      ERR_MQTT_COMMAND_MULTIPLE_INPUT : Word := 16#8001;   // Error - wrong operation - simultaneous input
      ERR_MQTT_COMMAND_PUBLISH_TOPIC_INVALID : Word := 16#8300;   // Error - publish topic empty or invalid
      ERR_MQTT_COMMAND_SUBSCRIBE_TOPIC_INVALID : Word := 16#8310;   // Error - subscribe topic empty or invalid
      ERR_MQTT_COMMAND_UNSUBSCRIBE_TOPIC_INVALID : Word := 16#8320;   // Error - unsubscribe topic empty or invalid
      ERR_MQTT_COMMAND_SEND_TIMEOUT : Word := 16#8650;   // Error - timeout while trying to sending data
      ERR_MQTT_CONNECT_TIMEOUT : Word := 16#8670;   // Error - timout while trying to connect via mqtt to broker
      MAX_BUFFER_LEN_RCV : UInt := 1459;   // Max. Buffer Len for TRCV
      MAX_BUFFER_LEN_SEND : UInt := 8191;   // Max. Buffer Len for TSEND on S7-1200/S7-1500
      EMPTY_BYTE : Byte := 16#00;   // Empty byte for initalisation
      NO_COMMAND : Byte := 16#00;   // No Command for Executing Publish, Subscribe, Unsubscribe
      EMPTY_STRING : String;   // Empty string for initalisation
      EMPTY_WSTRING : WString;   // Empty wstring for initalisation
      LEN_NULL : Int := 0;   // Integer 0 to compare length to zero
      INIT_UDINT_1 : UDInt := 1;   // Udint with value 1 for initalisation
      ARRAY_LEN_OFFSET_PLUS_1 : DInt := 1;   // Offset for array boundaries
      FIRST_CHARACTER : DInt := 1;   // First character in a character string
      ONE_DIMENSION : UDInt := 1;   // one dimensional array
      FIRST_ENCODING : DInt := 1;   // First encoding state while encoding messages
      SUBSEQUENT_ENCODING : DInt := 2;   // Followig encoding state while encoding messages if it takes multiple cycles
      ENCODE_DONE : DInt := 3;   // Last encoding state while encoding messages
      NOT_USED_NO_ENCODING : DInt := 5;   // No encoding state while encoding messages
      MSG_DECODE_STATE_NO_PROCESSING : DInt := 0;   // No message processing
      MSG_DECODE_STATE_TOPIC : DInt := 1;   // Message decoding state for topic
      MSG_DECODE_STATE_PAKET_ID_MSB : DInt := 2;   // Message decoding state for paket id msb
      MSG_DECODE_STATE_PAKET_ID_LSB : DInt := 3;   // Message decoding state for paket id lsb
      MSG_DECODE_STATE_PAYLOAD : DInt := 4;   // Message decoding state for paket payload
      MSG_DECODE_STATUS_NO_NEW_MSG : USInt := 0;   // Message decoding status if no new message was received
      MSG_DECODE_STATUS_NEW_MSG_OK : USInt := 1;   // Message decoding status if anew message was received
      MSG_DECODE_STATUS_TOPIC_TOO_LONG : USInt := 2;   // Message decoding status if new message was received bute topic does not fit it inout topic (too shoirt)
      MSG_DECODE_STATUS_PAYLOAD_TOO_LONG : USInt := 2;   // Message decoding status if new message was received bute payload does not fit it inout payload(too shoirt)
      MQTT_QOS_0 : UInt := 0;   // Saving mqtt qos 0
      MQTT_QOS_1 : UInt := 1;   // Saving mqtt qos 1
      MQTT_QOS_2 : UInt := 2;   // Saving mqtt qos 2
      REMAINING_LEN_3 : Byte := 16#03;   // Remaining len in bytes is 3
      REMAINING_LEN_2 : Byte := 16#02;   // Remaining len in bytes is 2
      REMAINIG_LEN_0 : Byte := 16#00;   // Remaining len in bytes is 0
      SUBSCRIBE_FAILURE : Byte := 16#80;   // Subscription failed flag.
      MQTT_NO_SESSION_PRESENT : Byte := 16#00;   // No session present indication
      KEEPALIVE_DISABLED : Time := t#0s;   // Mqtt keepalive set to 0s
      TSENDC_JOB_DONE : Word := 16#0000;   // Status of tsendc if job was successful
      TSENDC_COM_CLOSED : Word := 16#0003;   // Status of tsendc if connection closed
      TSENDC_EST_OK : Word := 16#7004;   // Status of tsendc if connection ok
      TSENDC_DISCONNECTED : Word := 16#7000;   // Status of tsendc if disconnected from broker
      UINT_CONST_1000 : UInt := 1000;   // Calculation to seconds
      TWO_SECONDS : UInt := 2000;   // Calculation by 2 seconds
      THREE_SECONDS : UInt := 3;   // Upper limit is 3 seconds
      UTF_1_BYTE_USED : USInt := 1;   // If utf uses 1 byte
      UTF_2_BYTE_USED : USInt := 2;   // If utf uses 2 byte
      UTF_3_BYTE_USED : USInt := 3;   // If utf uses 3 byte
      ONE_BYTE_LEN_INFO : UInt := 1;   // Adds one byte len info
      TWO_BYTE_LEN_INFO : UInt := 2;   // Adds two byte len info
      CONNECT_HEADER_10BYTE_LEN : UInt := 10;   // Connect header has always 10 byte minimum
      NO_RESPONSE : USInt := 0;   // If no response received from broker
      RESPONSE_GOOD : USInt := 1;   // If good response received from broker
      RESPONSE_PAKET_ID_INVALID : USInt := 2;   // If response received from broker but paket id invalid
      RESPONSE_SUBSCRIBE_FAILED : USInt := 3;   // If response received from broker but subscribption invalid
      MQTT_MSG_TYPE_CONNECT : Byte := 16#10;   // CONNECT MQTT Control Packet (see MQTT standard for more info)
      MQTT_MSG_TYPE_CONNACK : Byte := 16#20;   // CONNACK MQTT Control Packet (see MQTT standard for more info)
      MQTT_MSG_TYPE_DISCONNECT : Byte := 16#E0;   // DISCONNECT MQTT Control Packet (see MQTT standard for more info)
      MQTT_MSG_TYPE_PUBLISH : Byte := 16#30;   // PUBLISH MQTT Control Packet for QoS = 0 (see MQTT standard for more info)
      MQTT_MSG_TYPE_PUBACK : Byte := 16#40;   // PUBACK MQTT Control Packet (see MQTT standard for more info)
      MQTT_MSG_TYPE_PUBREC : Byte := 16#50;   // PUBREC MQTT Control Packet (see MQTT standard for more info)
      MQTT_MSG_TYPE_PUBREL : Byte := 16#62;   // PUBREL MQTT Control Packet (see MQTT standard for more info)
      MQTT_MSG_TYPE_PUBCOMP : Byte := 16#70;   // PUBCOM MQTT Control Packet (see MQTT standard for more info)
      MQTT_MSG_TYPE_SUBSCRIBE : Byte := 16#82;   // SUBSCRIBE MQTT Control Packet (see MQTT standard for more info)
      MQTT_MSG_TYPE_UNSUBSCRIBE : Byte := 16#A2;   // UNSUBSCRIBE MQTT Control Packet (see MQTT standard for more info)
      MQTT_MSG_TYPE_SUBACK : Byte := 16#90;   // SUBACK MQTT Control Packet (see MQTT standard for more info)
      MQTT_MSG_TYPE_UNSUBACK : Byte := 16#B0;   // UNSUBACK MQTT Control Packet (see MQTT standard for more info)
      MQTT_MSG_TYPE_PING : Byte := 16#C0;   // PING MQTT Control Packet (see MQTT standard for more info)
      MQTT_MSG_TYPE_PINGRESP : Byte := 16#D0;   // PINGRESP MQTT Control Packet (see MQTT standard for more info)
      MQTT_MSG_TYPE_RCV_PUB_MESSAGE : Byte := 16#30;   // PUBLISH MQTT Control Packet for QoS = 0 (see MQTT standard for more info)
      MQTT_MSG_TYPE_RCV_PUB_MESSAGE_QoS0 : Byte := 16#30;   // PUBLISH MQTT Control Packet for QoS = 0 (see MQTT standard for more info)
      MQTT_MSG_TYPE_RCV_PUB_MESSAGE_QoS1 : Byte := 16#32;   // PUBLISH MQTT Control Packet for QoS = 1 (see MQTT standard for more info)
      MQTT_MSG_TYPE_RCV_PUB_MESSAGE_QoS2 : Byte := 16#34;   // PUBLISH MQTT Control Packet for QoS = 2 (see MQTT standard for more info)
      MQTT_MSG_TYPE_RCV_PUB_MESSAGE_BAD : Byte := 16#36;   // PUBLISH MQTT Control Packet for QoS =1 and QoS=2 at the same time (see MQTT standard for more info)
      MQTT_MSG_DECODING : Byte := 16#FF;   // STATE to show that currently a message is being decoded
      MQTT_CONNACK_ACCEPTED : Byte := 16#00;   // Connect acknowledge flag in case no session present flag was not set
      BIT_MASK_HIGHBITS : Byte := 16#F0;   // MQTT Message Types only use High bits, so we only use High bits and ignore low bits
      BIT_MASK_QOS : Byte := 16#F6;   // A Bit Mask to only validate recieved Byte against QOS Value
      DEFAULT_VALUE_ZERO : Int := 0;   // DEFAULT Value for Variables that a ZERO Based
      SEND_LEN_MULTIPLIER_UDINT_128 : UDInt := 128;   // Default mulitplier to calculate package length
      MAX_ALLOWED_PAKET_SIZE : UDInt := 2097152;   // The highest amount of payload to be sent by mqtt paket
      DEFAULT_MULTIPLIER_BYTE_127 : Byte := 16#7F;   // Default mulitplier to calculate package length
      CONN_PROTOCOL_NAME_0 : Byte := 16#00;   // Protocol version for mqtt
      CONN_PROTOCOL_NAME_4 : Byte := 16#04;   // Protocol version for mqtt
      CONN_PROTOCOL_MQTT_VERSION_3_1_1 : Byte := 16#04;   // Protocol version for mqtt
   END_VAR
BEGIN
   REGION BLOCK INFO HEADER
     //===============================================================================
     // SIEMENS (c)Copyright 2023
     //-------------------------------------------------------------------------------
     // Title:        LMQTT_Client
     // Function:     This FB implements an MQTT client. A user can publish data and
     //               subscribe to topics to receive data.
     // Library:      LMQTT
     // Author:       Siemens Industry Online Support
     // Tested with:  CPU 1516-3 PN/DP FW 2.9
     // Engineering:  TIA Portal V17
     // Restrictions: --
     // Requirements: S7-1200 with firmware V4.4 or higher
     //               S7-1500 with firmware V2.0 or higher
     //-------------------------------------------------------------------------------
     // Change log table:
     // Version  | Date       | Expert in charge       | Changes applied
     //----------|------------|------------------------|------------------------------
     // 04.00.05 | 2024-06-05 | Online Support         | Fixed ActivateSecureConn reset
     // 04.00.04 | 2024-04-09 | Online Support         | Allowed lastWill without payload
     // 04.00.03 | 2024-02-12 | Online Support         | Improved evaluation of broker address
     // 04.00.02 | 2023-09-05 | Online Support         | Fixed bug that edge on publish/subscribe while PING is saved
     // 04.00.01 | 2023-08-30 | Online Support         | Fixed bug at TRCV and ConnID
     // 04.00.00 | 2023-08-04 | Online Support         | Broker can be addresses with hostname or IP address using one parameter
     //                                                | Reordered interface
     //                                                | Fixed bug at publish with QoS = 2
     // 03.00.05 | 2023-02-23 | Online Support         | Fixed bug that in rare situations no new commands were accepted
     // 03.00.04 | 2022-06-09 | Online Support         | Fixed bug that done was not set if input was reset
     // 03.00.03 | 2021-05-07 | Online Support         | Minor bug fixes
     // 03.00.00 | 2020-11-04 | Online Support         | New block interface with major improvements
     // 02.02.02 | 2020-03-16 | Online Support         | Improved issue with validateSubjectAlternateNameOfServer not setting correct bit
     // 02.02.01 | 2019-12-03 | Online Support         | Update to V16 and fusion with S7-1200 Lib
     // 02.01.00 | 2019-11-10 | Online Support         | Minor connection improvements. Updated some comments
     // 02.00.00 | 2018-06-04 | Online Support         | Added DNS support and Subscribe to topics
     // 01.00.00 | 2017-06-06 | Online Support         | First released version
     //===============================================================================
   END_REGION

   #tempEnable := #enable; // Work with temporary value / create process image
   #tempPublish := #publish;  // Work with temporary value / create process image - only checked when MQTT is connected
   #tempSubscribe := #subscribe;  // Work with temporary value / create process image - only checked when MQTT is connected
   #tempUnsubscribe := #unsubscribe;  // Work with temporary value / create process image - only checked when MQTT is connected


   REGION OUC_BLOCK_CALLS
     //Only call if FB is processing
     IF #statStatus <> #STATUS_NO_CALL THEN
       // Connect and send
       IF #statConnParam.isQDN = TRUE THEN // Call if host is a domain name
         #instTsendC(REQ     := #statTsendcReq,
                     CONT    := #statTsendcEnable,
                     LEN     := #statTsendcLen,
                     DONE    => #tempTsendcDone,
                     BUSY    => #tempTsendcBusy,
                     ERROR   => #tempTsendcError,
                     STATUS  => #tempTsendcStatus,
                     CONNECT := #statConnParam.paramQDN,
                     DATA    := #statSendBuffer);

       ELSE
         #instTsendC(REQ     := #statTsendcReq,
                     CONT    := #statTsendcEnable,
                     LEN     := #statTsendcLen,
                     DONE    => #tempTsendcDone,
                     BUSY    => #tempTsendcBusy,
                     ERROR   => #tempTsendcError,
                     STATUS  => #tempTsendcStatus,
                     CONNECT := #statConnParam.paramIP,
                     DATA    := #statSendBuffer);
       END_IF;

       // Receive only when TCP operating
       #instTrcv(EN_R     := (#statFBState = #FB_STATE_OPERATING_MONITOR_TCP),
                 ID       := #statConnParam.paramQDN.ConnPara.ID,
                 ADHOC    := true,
                 NDR      => #tempTrcvNdr,
                 BUSY     => #tempTrcvBusy,
                 ERROR    => #tempTrcvError,
                 STATUS   => #tempTrcvStatus,
                 RCVD_LEN => #tempTrcvRcvdLen,
                 DATA     := #statRcvBuffer);

       //Monitor Time out
       #instTimerCommandWatchdog.TON(IN := #statEnableTimerCommandWatchdog,
                                     PT := #timeOut);
       //Mqtt Keepalive Timer
       #instMqttKeepAliveTimer.TON(IN := #statEnableMqttKeepAliveTimer,
                                   PT := #statMqttKeepAliveTime);
     END_IF;
   END_REGION

   REGION ENABLING/DISABLING_FUNCTION_BLOCK
     IF (#tempEnable = TRUE) AND (#statStatus = #STATUS_NO_CALL) THEN // Enable FB
       // First call; initialize FB
       #statValid := TRUE;
       #statBusy := TRUE;
       #statError := FALSE;
       #statDone := FALSE;
       #statErrorUserCleared := FALSE;
       #statErrorAutoCleared := FALSE;
       #statStatus := #STATUS_FIRST_CALL;
       #statSubfunctionStatus := #STATUS_JOB_EXECUTED;
       #statFBErrorState := 0;
       #diagnostics := #statEmptyDiagnostics;
       #statDisablingCompleted := FALSE;
       // State machine - start functionality
       #statFBState := #FB_STATE_VALIDATE_INPUT;

       // Initialize functionality: reset of variables, diagnostics, etc.
       #statPublishOld := FALSE;
       #statSubscribeOld := FALSE;
       #statUnsubscribeOld := FALSE;
       #statConnParam.isQDN := FALSE;
       #statTsendcReq := FALSE;
       #statTsendcEnable := FALSE;
       #statTsendcLen := 0;
       #statEnableTimerCommandWatchdog := FALSE;
       #statEnableMqttKeepAliveTimer := FALSE;
       #statMqttKeepAliveTime := #KEEPALIVE_DISABLED;
       #statMqttKeepAliveUsed := FALSE;
       #statSendBufferPos := 0;
       #statPaketHeaderEncodeDone := FALSE;
       #statSendPaketTotalRemLen := 0;
       #statEncodedRemPaketLenAsByte := #EMPTY_BYTE;
       #statClientIdPos := 0;
       #statClientIdEncodeState := 0;
       #statClientIdLenUtf8Encoded := 0;
       #statUserNamePos := 0;
       #statUserNameEncodeState := #FIRST_ENCODING;
       #statUsernameLenUtf8Encoded := 0;
       #statPasswordPos := 0;
       #statPasswordEncodeState := #FIRST_ENCODING;
       #statPasswordLenUtf8Encoded := 0;
       #statWillQos := 0;
       #statWillRetain := FALSE;
       #statWillMessageCnt := 0;
       #statWillMessagePos := 0;
       #statWillMessageEncodeState := #FIRST_ENCODING;
       #statWillTopicLenUtf8Encoded := 0;
       #statWillTopicPos := 0;
       #statWillTopicEncodeState := #FIRST_ENCODING;
       #statPaketId := 0;
       #statPublishTopicLenUtf8Encoded := 0;
       #statPublishQos := 0;
       #statPublishMessageCnt := 0;
       #statPublishTopicEncodeState := #FIRST_ENCODING;
       #statPublishTopicPos := 0;
       #statPaketIdEncoded := FALSE;
       #statPublishEncodeMessageState := #FIRST_ENCODING;
       #statPublishMessagePos := 0;
       #statSubscribeQos := 0;
       #statSubscribeQosEncoded := FALSE;
       #statSubscribeTopicPos := 0;
       #statSubscribeTopicEncodeState := #FIRST_ENCODING;
       #statSubscribeTopicLenUtf8Encoded := 0;
       #statUnsubscribeTopicPos := 0;
       #statUnsubscribeTopicEncodeState := #FIRST_ENCODING;
       #statUnsubscribeTopicLenUtf8Encoded := 0;
       #statRcvMsgQoS := 0;
       #statRcvMsgTotalLen := 0;
       #statRcvMsgTopicLen := 0;
       #statRcvMsgPayloadLen := 0;
       #statRcvMsgPaketId := 0;
       #statRcvMsgTopicPos := 0;
       #statRcvMsgPayloadPos := 0;
       #statRcvMsgDecodeState := #MSG_DECODE_STATE_NO_PROCESSING;
       #statRcvMsgInternalStatus := 0;
       #statRcvMsgStatus := 0;
       #statRcvMsgDataLen := 0;
       #statSendPubAckMsg := FALSE;

       // Initialize functionality: call subsidiary FBs with FALSE
       FILL_BLK(IN    := #EMPTY_BYTE,
                COUNT := #MAX_BUFFER_LEN_SEND,
                OUT   => #statSendBuffer[0]);
       FILL_BLK(IN    := #EMPTY_BYTE,
                COUNT := #MAX_BUFFER_LEN_RCV,
                OUT   => #statRcvBuffer[0]);
       RESET_TIMER(#instTimerCommandWatchdog);
       RESET_TIMER(#instMqttKeepAliveTimer);

       // INIT SUB STATE MACHINES
       #statMqttConnectState := #MQTT_CONNECT_STATE_NO_PROCESSING;
       #statMqttCommandState := #MQTT_COMMAND_STATE_NO_PROCESSING;
       #statRcvMsgDecodeState := #MSG_DECODE_STATE_NO_PROCESSING;

     ELSIF (#tempEnable = FALSE) AND (#statEnableOld = TRUE) THEN // Disable FB 
       #statFBState := #FB_STATE_DISABLING;
     ELSIF (#statStatus = #STATUS_FIRST_CALL) THEN // Set status identifier of subsequent call
       #statStatus := #STATUS_SUBSEQUENT_CALL;
     END_IF;

     // Edge detection 'enable' input
     #statEnableOld := #tempEnable;
   END_REGION ENABLING/DISABLING

   IF (#statStatus = #STATUS_NO_CALL) THEN // Nothing to do -> End here to reduce "system load"
     RETURN;
   END_IF;

   REGION STATE_MACHINE_FUNCTION_BLOCK_TCP
     CASE #statFBState OF // State machine of FB
       #FB_STATE_NO_PROCESSING: // No processing active (Note: this state must always be present and left empty)
         ;

       #FB_STATE_VALIDATE_INPUT: // Enabling active
         REGION EVALUATE CONNECTION PARAMETERS
           // Determine if host is domain name or IP address
           #statConnParam.isQDN := NOT "IsIPAddress"(address := #connParam.broker, ipAddress => #statConnParam.paramIP.ConnPara.RemoteAddress);

           IF #statConnParam.isQDN THEN // Broker address is a hostname
             IF #connParam.broker[LEN(#connParam.broker)] = '.' THEN
               #statConnParam.paramQDN.ConnPara.RemoteQDN := #connParam.broker;
             ELSE
               #statConnParam.paramQDN.ConnPara.RemoteQDN := CONCAT(IN1 := #connParam.broker, IN2 := '.');
             END_IF;

             #statConnParam.paramQDN.ConnPara.InterfaceId := #connParam.hwId;
             #statConnParam.paramQDN.ConnPara.ID := #connParam.connId;
             #statConnParam.paramQDN.ConnPara.ActiveEstablished := TRUE;
             #statConnParam.paramQDN.ConnPara.RemotePort := #connParam."port";
           ELSE // Broker address is an IP address
             #statConnParam.paramIP.ConnPara.InterfaceId := #connParam.hwId;
             #statConnParam.paramIP.ConnPara.ID := #statConnParam.paramQDN.ConnPara.ID := #connParam.connId;
             #statConnParam.paramIP.ConnPara.ActiveEstablished := TRUE;
             #statConnParam.paramIP.ConnPara.RemotePort := #connParam."port";
           END_IF;

           IF #connParam.tls.enableTls THEN
             IF #statConnParam.isQDN THEN
               #statConnParam.paramQDN.ActivateSecureConn := TRUE;
               #statConnParam.paramQDN.ExtTLSCapabilities.%X0 := #connParam.tls.validateServerIdentity;
               #statConnParam.paramQDN.TLSServerCertRef := #connParam.tls.brokerCert;
               #statConnParam.paramQDN.TLSClientCertRef := #connParam.tls.clientCert;
             ELSE
               #statConnParam.paramIP.ActivateSecureConn := TRUE;
               #statConnParam.paramIP.ExtTLSCapabilities.%X0 := #connParam.tls.validateServerIdentity;
               #statConnParam.paramIP.TLSServerCertRef := #connParam.tls.brokerCert;
               #statConnParam.paramIP.TLSClientCertRef := #connParam.tls.clientCert;
             END_IF;
           ELSE
             IF #statConnParam.isQDN THEN
               #statConnParam.paramQDN.ActivateSecureConn := FALSE;

             ELSE
               #statConnParam.paramIP.ActivateSecureConn := FALSE;

             END_IF;
           END_IF;
         END_REGION EVALUATE CONNECTION PARAMETERS

         REGION FB_VALIDATE_INPUT     
           //Check Input variables:
           #tempMaxWillMsgLen := ABS(UPPER_BOUND(ARR := #willMsgPayload, DIM := #ONE_DIMENSION) - LOWER_BOUND(ARR := #willMsgPayload, DIM := #ONE_DIMENSION)) + #ARRAY_LEN_OFFSET_PLUS_1;

           //Check Client ID len Must be > 0 
           IF LEN(#clientIdentifier) <= #LEN_NULL THEN
             #statStatus := #ERR_CLIENT_ID_NULL; // Set correct status that identifies error clearly
             #statSubfunctionStatus := #ERR_CLIENT_ID_NULL; // Status or return value of called FBs, FCs and system blocks
             #statFBErrorState := #statFBState; // Set error state number for diagnostic 
             #statErrorUserCleared := TRUE;
             //verify Will next
           ELSIF #tempMaxWillMsgLen < #willMsgLen THEN
             #statStatus := #ERR_CNT_EXCEEDS_ARRAY_DIMENSION; // Set correct status that identifies error clearly
             #statSubfunctionStatus := #ERR_CNT_EXCEEDS_ARRAY_DIMENSION; // Status or return value of called FBs, FCs and system blocks
             #statFBErrorState := #statFBState; // Set error state number for diagnostic 
             #statErrorUserCleared := TRUE;
             ///CHECK WILL QOS
           ELSIF #qos > #MQTT_QOS_2 THEN
             #statStatus := #ERR_QOS_INVALID; // Set correct status that identifies error clearly
             #statSubfunctionStatus := #ERR_QOS_INVALID; // Status or return value of called FBs, FCs and system blocks
             #statFBErrorState := #statFBState; // Set error state number for diagnostic 
             #statErrorUserCleared := TRUE;
           ELSIF (#connParam.keepAlive < #THREE_SECONDS) // IF Set to 1 or 2 seconds..
             AND (#connParam.keepAlive > 0)
           THEN
             #statStatus := #ERR_KEEPALIVE_INVALID; // Set correct status that identifies error clearly
             #statSubfunctionStatus := #ERR_KEEPALIVE_INVALID; // Status or return value of called FBs, FCs and system blocks
             #statFBErrorState := #statFBState; // Set error state number for diagnostic 
             #statErrorUserCleared := TRUE;
           ELSE
             //Set Params for connection
             //Set Client Id
             #statWillQos := #qos;
             //set Retain
             #statWillRetain := #retain;
             // Will message cnt
             #statWillMessageCnt := #willMsgLen;

             //Keepalive
             IF #connParam.keepAlive = 0 THEN
               #statMqttKeepAliveUsed := FALSE;
             ELSE
               #statMqttKeepAliveUsed := TRUE;
               //KeepAliveTImer is set to ((Keep Alive converted to seconds) - 2s)
               #statMqttKeepAliveTime := UINT_TO_TIME((#connParam.keepAlive * #UINT_CONST_1000 - #TWO_SECONDS));
             END_IF;

             //rdy to enable TCON
             #statTsendcEnable := TRUE;
             #statEnableTimerCommandWatchdog := TRUE;
             #statFBState := #FB_STATE_TCP_CONNECTING;
           END_IF;
         END_REGION FB_VALIDATE_INPUT

       #FB_STATE_TCP_CONNECTING: //Wait for TCP to be established
         REGION FB_TCP_CONNECTING
           //Check process:
           IF #tempTsendcError = TRUE THEN //when error:
             #statTsendcEnable := FALSE; //disable TsendC
             #statEnableTimerCommandWatchdog := FALSE;
             #statStatus := #ERR_TCON_FAILED; // Set correct status that identifies error clearly
             #statSubfunctionStatus := #tempTsendcStatus; // Status or return value of called FBs, FCs and system blocks
             #statFBErrorState := #statFBState; // Set error state number for diagnostic 
             #statErrorUserCleared := TRUE;
           ELSIF #tempTsendcStatus = #TSENDC_EST_OK THEN //when successfull:
             //     Communication connection established.
             #statEnableTimerCommandWatchdog := FALSE;
             //Monitor Connection
             #statFBState := #FB_STATE_OPERATING_MONITOR_TCP;
             // Begin MQTT Connection
             #statMqttConnectState := #MQTT_CONNECT_STATE_BUILD_PAKET;
             //set status
             #statStatus := #STATUS_MQTT_CONNECTING;
           ELSIF #instTimerCommandWatchdog.Q THEN
             #statTsendcEnable := FALSE; //disable TsendC
             #statEnableTimerCommandWatchdog := FALSE;
             #statStatus := #ERR_TCON_TIMEOUT; // Set correct status that identifies error clearly
             #statSubfunctionStatus := #ERR_TCON_TIMEOUT; // Status or return value of called FBs, FCs and system blocks
             #statFBErrorState := #statFBState; // Set error state number for diagnostic 
             #statErrorUserCleared := TRUE;
           END_IF;
         END_REGION FB_TCP_CONNECTING
       #FB_STATE_OPERATING_MONITOR_TCP: // Processing active
         REGION FB_OPERATING_MONITOR_TCP
           //Reset Status on Msg Output - will be set when a new message is completly processed and ready at outputs.
           #statRcvMsgStatus := #MSG_DECODE_STATUS_NO_NEW_MSG;
           //Reset TsendC Req from last  cycle Request:

           #statTsendcReq := FALSE;

           //Monitor Connection - if disconnect occured:
           IF ((#tempTsendcStatus > #TSENDC_COM_CLOSED AND #tempTsendcStatus < #TSENDC_EST_OK) //Status connection interupt
             OR #tempTsendcError = TRUE) // Or error
             AND #tempTrcvNdr = FALSE // And no new data (to see if broker send information why connection was interrupted)
           THEN
             REGION CONNECTION_INTERRUPTED
               //Status reconnecting
               //SET MQTT to no operation
               #statMqttConnectState := #MQTT_CONNECT_STATE_NO_PROCESSING;
               #statMqttCommandState := #MQTT_COMMAND_STATE_NO_PROCESSING;
               #statRcvMsgDecodeState := #MSG_DECODE_STATE_NO_PROCESSING;
               //Reset Pub ack
               #statSendPubAckMsg := FALSE;
               //reset Done bit if still set, regardless of input:
               #statDone := FALSE;
               //reset Watchdog
               #statEnableTimerCommandWatchdog := FALSE;
               // reset headerEncode
               #statPaketHeaderEncodeDone := FALSE;
               //set error  information
               #statStatus := #ERR_TCP_RECONNECTING; // Set correct status that identifies error clearly
               #statSubfunctionStatus := #tempTsendcStatus;// Status or return value of called FBs, FCs and system blocks
               #statFBErrorState := #statFBState; // Set error state number for diagnostic 
               #statErrorAutoCleared := TRUE;
               //Wait for reconect - next state
               #statFBState := #FB_STATE_TCP_RECONNECTING;
             END_REGION REGION CONNECTION_INTERRUPTED
           ELSE
             //Connection is OK
             //Sending and receiving works 
             //Check Trcv Buffer for new Data
             IF #tempTrcvNdr THEN
               REGION TRCV_NEW_DATA
                 //Evaluate the TrcvBuffer, reset buffer pos to start
                 #tempTrcvBufferPos := 0;
                 // Parse the whole RCV Buffer
                 WHILE #tempTrcvBufferPos < (UDINT_TO_DINT(#tempTrcvRcvdLen)) DO
                   // Parse the whole RCV Buffer, check wether header or decoding
                   IF #statRcvMsgDecodeState = #MSG_DECODE_STATE_NO_PROCESSING THEN
                     //If no decoding is in progress, look for new message header
                     #tempRcvMsgTypeCase := #statRcvBuffer[#tempTrcvBufferPos] AND #BIT_MASK_HIGHBITS;
                   ELSE
                     //decode is in progress, go directly to decoding
                     #tempRcvMsgTypeCase := #MQTT_MSG_DECODING;
                   END_IF;

                   CASE #tempRcvMsgTypeCase OF
                     #MQTT_MSG_TYPE_CONNACK:  // Statement section case 1
                       REGION RECEIVED_CONACK_PACKET    
                         #tempTrcvBufferPos += 1;
                         IF #statRcvBuffer[#tempTrcvBufferPos] = #REMAINING_LEN_2 //remainng Length must be 2;
                         THEN //
                           #tempTrcvBufferPos += 1;
                           //byte one is 0000 000X where X is if Session was set // so depending on clean session or not  evaluate answer of server
                           IF #statRcvBuffer[#tempTrcvBufferPos] = #MQTT_NO_SESSION_PRESENT THEN
                             #tempTrcvBufferPos += 1;
                             //VALID Answer, check code
                             IF #statRcvBuffer[#tempTrcvBufferPos] = #MQTT_CONNACK_ACCEPTED
                             THEN
                               //All good
                               #tempTrcvBufferPos += 1;
                               #tempMqttConnAckRcvStatus := #RESPONSE_GOOD; //evaluate in MQTT StateMachine Below the response
                             ELSE
                               //NOT VALID CONNACK from server shows session has a bad return code
                               #statStatus := #ERR_MQTT_CONNACK_RETURN_CODE_INVALID; // Set correct status that identifies error clearly
                               #statSubfunctionStatus := #statRcvBuffer[#tempTrcvBufferPos]; // Status or return value of called FBs, FCs and system blocks
                               #statFBErrorState := #statFBState; // Set error state number for diagnostic 
                               #statErrorUserCleared := TRUE;
                               // Exit loop
                               EXIT;
                             END_IF;
                           ELSE
                             //NOT VALID, CONNACK from server shows session present
                             #statStatus := #ERR_MQTT_CONNACK_INVALID_SESSION_FLAG; // Set correct status that identifies error clearly
                             #statSubfunctionStatus := #ERR_MQTT_CONNACK_INVALID_SESSION_FLAG; // Status or return value of called FBs, FCs and system blocks
                             #statFBErrorState := #statFBState; // Set error state number for diagnostic 
                             #statErrorUserCleared := TRUE;
                             // Exit loop
                             EXIT;
                           END_IF;
                         ELSE // We got a CONNACK paket, but remaining length was not 2 (Error)
                           #statStatus := #ERR_MQTT_REM_LEN_INVALID; // Set correct status that identifies error clearly
                           #statSubfunctionStatus := #ERR_MQTT_REM_LEN_INVALID; // Status or return value of called FBs, FCs and system blocks
                           #statFBErrorState := #statFBState; // Set error state number for diagnostic 
                           #statErrorUserCleared := TRUE;
                           // Exit loop
                           EXIT;
                         END_IF;
                       END_REGION RECEIVED_CONACK_PACKET 

                     #MQTT_MSG_TYPE_PINGRESP:
                       REGION RECEIVED_PINGRESP_PACKET
                         #tempTrcvBufferPos += 1;
                         IF #statRcvBuffer[#tempTrcvBufferPos] = #REMAINIG_LEN_0 //remainng Length must be 0;
                         THEN
                           #tempTrcvBufferPos += 1;
                           #tempMqttPingRspRcv := #RESPONSE_GOOD; //evaluate in MQTT StateMachine Below the response
                         ELSE// We got a Pingrsp paket, but remaining length was not 0 (Error)
                           #statStatus := #ERR_MQTT_REM_LEN_INVALID; // Set correct status that identifies error clearly
                           #statSubfunctionStatus := #ERR_MQTT_REM_LEN_INVALID; // Status or return value of called FBs, FCs and system blocks
                           #statFBErrorState := #statFBState; // Set error state number for diagnostic 
                           #statErrorUserCleared := TRUE;
                           // Exit loop
                           EXIT;
                         END_IF;
                       END_REGION RECEIVED_PINGRESP_PAKET

                     #MQTT_MSG_TYPE_PUBACK:
                       REGION RECEIVED_PUBACK_PAKET
                         #tempTrcvBufferPos += 1;
                         IF #statRcvBuffer[#tempTrcvBufferPos] = #REMAINING_LEN_2 //remainng Length must be 2;
                         THEN //
                           #tempTrcvBufferPos += 1;
                           #tempWordForSliceAddress := UINT_TO_WORD(#statPaketId);
                           IF #statRcvBuffer[#tempTrcvBufferPos] = #tempWordForSliceAddress.%B1 THEN
                             #tempTrcvBufferPos += 1;
                             IF #statRcvBuffer[#tempTrcvBufferPos] = #tempWordForSliceAddress.%B0 THEN
                               #tempTrcvBufferPos += 1;
                               #tempMqttPubAckRcv := #RESPONSE_GOOD;
                             ELSE
                               #tempTrcvBufferPos += 1;
                               #tempMqttPubAckRcv := #RESPONSE_PAKET_ID_INVALID;
                             END_IF;
                           ELSE
                             #tempTrcvBufferPos += 1;
                             #tempMqttPubAckRcv := #RESPONSE_PAKET_ID_INVALID;
                           END_IF;
                         ELSE
                           #statStatus := #ERR_MQTT_REM_LEN_INVALID; // Set correct status that identifies error clearly
                           #statSubfunctionStatus := #ERR_MQTT_REM_LEN_INVALID; // Status or return value of called FBs, FCs and system blocks
                           #statFBErrorState := #statFBState; // Set error state number for diagnostic 
                           #statErrorUserCleared := TRUE;
                           // Exit loop
                           EXIT;
                         END_IF;
                       END_REGION RECEIVED_PUBACK_PAKET

                     #MQTT_MSG_TYPE_PUBREC:
                       REGION RECEIVED_PUBREC_PAKET
                         #tempTrcvBufferPos += 1;
                         IF #statRcvBuffer[#tempTrcvBufferPos] = #REMAINING_LEN_2 //remainng Length must be 2;
                         THEN //
                           #tempTrcvBufferPos += 1;
                           #tempWordForSliceAddress := UINT_TO_WORD(#statPaketId);
                           IF #statRcvBuffer[#tempTrcvBufferPos] = #tempWordForSliceAddress.%B1 THEN
                             #tempTrcvBufferPos += 1;
                             IF #statRcvBuffer[#tempTrcvBufferPos] = #tempWordForSliceAddress.%B0 THEN
                               #tempTrcvBufferPos += 1;
                               #statMqttPubRecRcv := #RESPONSE_GOOD;
                             ELSE
                               #tempTrcvBufferPos += 1;
                               #statMqttPubRecRcv := #RESPONSE_PAKET_ID_INVALID;
                             END_IF;
                           ELSE
                             #tempTrcvBufferPos += 1;
                             #statMqttPubRecRcv := #RESPONSE_PAKET_ID_INVALID;
                           END_IF;
                         ELSE
                           #statStatus := #ERR_MQTT_REM_LEN_INVALID; // Set correct status that identifies error clearly
                           #statSubfunctionStatus := #ERR_MQTT_REM_LEN_INVALID; // Status or return value of called FBs, FCs and system blocks
                           #statFBErrorState := #statFBState; // Set error state number for diagnostic 
                           #statErrorUserCleared := TRUE;
                           // Exit loop
                           EXIT;
                         END_IF;
                       END_REGION RECEIVED_PUBREC_PAKET

                     #MQTT_MSG_TYPE_PUBCOMP:
                       REGION RECEIVED_PUBCOMP_PAKET
                         #tempTrcvBufferPos += 1;
                         IF #statRcvBuffer[#tempTrcvBufferPos] = #REMAINING_LEN_2 //remainng Length must be 2;
                         THEN //
                           #tempTrcvBufferPos += 1;
                           #tempWordForSliceAddress := UINT_TO_WORD(#statPaketId);
                           IF #statRcvBuffer[#tempTrcvBufferPos] = #tempWordForSliceAddress.%B1 THEN
                             #tempTrcvBufferPos += 1;
                             IF #statRcvBuffer[#tempTrcvBufferPos] = #tempWordForSliceAddress.%B0 THEN
                               #tempTrcvBufferPos += 1;
                               #tempMqttPubCompRcv := #RESPONSE_GOOD;

                             ELSE
                               #tempTrcvBufferPos += 1;
                               #tempMqttPubCompRcv := #RESPONSE_PAKET_ID_INVALID;

                             END_IF;
                           ELSE
                             #tempTrcvBufferPos += 1;
                             #tempMqttPubCompRcv := #RESPONSE_PAKET_ID_INVALID;

                           END_IF;
                         ELSE
                           #statStatus := #ERR_MQTT_REM_LEN_INVALID; // Set correct status that identifies error clearly
                           #statSubfunctionStatus := #ERR_MQTT_REM_LEN_INVALID; // Status or return value of called FBs, FCs and system blocks
                           #statFBErrorState := #statFBState; // Set error state number for diagnostic 
                           #statErrorUserCleared := TRUE;
                           // Exit loop
                           EXIT;
                         END_IF;
                       END_REGION RECEIVED_PUBCOMP_PAKET

                     #MQTT_MSG_TYPE_SUBACK:
                       REGION RECEIVED_SUBACK_PAKET
                         #tempTrcvBufferPos += 1;
                         IF #statRcvBuffer[#tempTrcvBufferPos] = #REMAINING_LEN_3 //remainng Length must be 3;
                         THEN //
                           #tempTrcvBufferPos += 1;
                           #tempWordForSliceAddress := UINT_TO_WORD(#statPaketId);
                           IF #statRcvBuffer[#tempTrcvBufferPos] = #tempWordForSliceAddress.%B1 THEN
                             #tempTrcvBufferPos += 1;
                             IF #statRcvBuffer[#tempTrcvBufferPos] = #tempWordForSliceAddress.%B0 THEN
                               #tempTrcvBufferPos += 1;
                               IF #statRcvBuffer[#tempTrcvBufferPos] = #SUBSCRIBE_FAILURE THEN
                                 #tempTrcvBufferPos += 1;
                                 #tempMqttSubAckRcv := #RESPONSE_SUBSCRIBE_FAILED;
                               ELSE
                                 #tempTrcvBufferPos += 1;
                                 #tempMqttSubAckRcv := #RESPONSE_GOOD;
                               END_IF;
                             ELSE
                               #tempTrcvBufferPos += 1;
                               #tempMqttSubAckRcv := #RESPONSE_PAKET_ID_INVALID;
                             END_IF;
                           ELSE
                             #tempTrcvBufferPos += 1;
                             #tempMqttSubAckRcv := #RESPONSE_PAKET_ID_INVALID;
                           END_IF;
                         ELSE
                           #statStatus := #ERR_MQTT_REM_LEN_INVALID; // Set correct status that identifies error clearly
                           #statSubfunctionStatus := #ERR_MQTT_REM_LEN_INVALID; // Status or return value of called FBs, FCs and system blocks
                           #statFBErrorState := #statFBState; // Set error state number for diagnostic 
                           #statErrorUserCleared := TRUE;
                           // Exit loop
                           EXIT;
                         END_IF;
                       END_REGION RECEIVED_SUBACK_PAKET

                     #MQTT_MSG_TYPE_UNSUBACK:
                       REGION RECEIVED_UNSUBACK_PAKET
                         #tempTrcvBufferPos += 1;
                         IF #statRcvBuffer[#tempTrcvBufferPos] = #REMAINING_LEN_2 //remainng Length must be 2;
                         THEN //
                           #tempTrcvBufferPos += 1;
                           #tempWordForSliceAddress := UINT_TO_WORD(#statPaketId);
                           IF #statRcvBuffer[#tempTrcvBufferPos] = #tempWordForSliceAddress.%B1 THEN
                             #tempTrcvBufferPos += 1;
                             IF #statRcvBuffer[#tempTrcvBufferPos] = #tempWordForSliceAddress.%B0 THEN
                               #tempTrcvBufferPos += 1;
                               #tempMqttUnSubAckRcv := #RESPONSE_GOOD;
                             ELSE
                               #tempTrcvBufferPos += 1;
                               #tempMqttUnSubAckRcv := #RESPONSE_PAKET_ID_INVALID;
                             END_IF;
                           ELSE
                             #tempTrcvBufferPos += 1;
                             #tempMqttUnSubAckRcv := #RESPONSE_PAKET_ID_INVALID;
                           END_IF;
                         ELSE
                           #statStatus := #ERR_MQTT_REM_LEN_INVALID; // Set correct status that identifies error clearly
                           #statSubfunctionStatus := #ERR_MQTT_REM_LEN_INVALID; // Status or return value of called FBs, FCs and system blocks
                           #statFBErrorState := #statFBState; // Set error state number for diagnostic 
                           #statErrorUserCleared := TRUE;
                           // Exit loop
                           EXIT;
                         END_IF;
                       END_REGION RECEIVED_UNSUBACK_PAKET

                     #MQTT_MSG_TYPE_RCV_PUB_MESSAGE:
                       REGION RECEIVED_PUBLISH_PAKET_FROM_BROKER
                         //Received a message, start process.
                         //init
                         #tempMultiplierToDecode := #INIT_UDINT_1;
                         #statRcvMsgInternalStatus := #MSG_DECODE_STATUS_NO_NEW_MSG;
                         #statRcvMsgTotalLen := 0;
                         #statRcvMsgTopicLen := 0;
                         #statRcvMsgPayloadLen := 0;
                         //Check and store QoS for later use
                         IF (#statRcvBuffer[#tempTrcvBufferPos] AND #BIT_MASK_QOS) = #MQTT_MSG_TYPE_RCV_PUB_MESSAGE_QoS0
                         THEN
                           #statRcvMsgQoS := #MQTT_QOS_0;
                         ELSIF (#statRcvBuffer[#tempTrcvBufferPos] AND #BIT_MASK_QOS) = #MQTT_MSG_TYPE_RCV_PUB_MESSAGE_QoS1
                         THEN
                           #statRcvMsgQoS := #MQTT_QOS_1;
                         ELSIF (#statRcvBuffer[#tempTrcvBufferPos] AND #BIT_MASK_QOS) = #MQTT_MSG_TYPE_RCV_PUB_MESSAGE_QoS2
                         THEN
                           #statRcvMsgQoS := #MQTT_QOS_2;
                         ELSIF (#statRcvBuffer[#tempTrcvBufferPos] AND #BIT_MASK_QOS) = #MQTT_MSG_TYPE_RCV_PUB_MESSAGE_BAD
                         THEN
                           #statStatus := #ERR_MQTT_MALFORMED_QOS_RECEIVED; // Set correct status that identifies error clearly
                           #statSubfunctionStatus := #ERR_MQTT_MALFORMED_QOS_RECEIVED; // Status or return value of called FBs, FCs and system blocks
                           #statFBErrorState := #statFBState; // Set error state number for diagnostic 
                           #statErrorUserCleared := TRUE;
                           // Exit loop
                           EXIT;
                         END_IF;

                         //Calculate total publish len (topic,paketid,payload)
                         REPEAT
                           #tempTrcvBufferPos += 1; //Increment
                           #statRcvMsgTotalLen += BYTE_TO_UDINT((#statRcvBuffer[#tempTrcvBufferPos] AND #DEFAULT_MULTIPLIER_BYTE_127)) * #tempMultiplierToDecode;
                           #tempMultiplierToDecode *= #SEND_LEN_MULTIPLIER_UDINT_128;
                           IF (#tempMultiplierToDecode > #MAX_ALLOWED_PAKET_SIZE)
                           THEN//Throw error here // Malformed remain length.
                             #statStatus := #ERR_MQTT_REM_LEN_INVALID; // Set correct status that identifies error clearly
                             #statSubfunctionStatus := #ERR_MQTT_REM_LEN_INVALID; // Status or return value of called FBs, FCs and system blocks
                             #statFBErrorState := #statFBState; // Set error state number for diagnostic 
                             #statErrorUserCleared := TRUE;
                             // Exit loop
                             EXIT;
                           END_IF;
                         UNTIL ((#statRcvBuffer[#tempTrcvBufferPos] AND UDINT_TO_BYTE(#SEND_LEN_MULTIPLIER_UDINT_128)) = 0)
                         END_REPEAT;
                         #tempTrcvBufferPos += 1; //Increment
                         //#statIncPaketRemLen contains total paket len
                         //Save Topic Len
                         #tempWordForSliceAddress.%B1 := #statRcvBuffer[#tempTrcvBufferPos]; //MSB
                         #tempTrcvBufferPos += 1; //Increment
                         #tempWordForSliceAddress.%B0 := #statRcvBuffer[#tempTrcvBufferPos]; //LSB
                         #tempTrcvBufferPos += 1; //Increment
                         #statRcvMsgTopicLen := WORD_TO_UINT(#tempWordForSliceAddress);
                         //Set Payload len
                         IF #statRcvMsgQoS = #MQTT_QOS_0 THEN
                           //Payload Len is total Len minus topic len minus topic len info 
                           #statRcvMsgPayloadLen := #statRcvMsgTotalLen - #statRcvMsgTopicLen - #TWO_BYTE_LEN_INFO;
                         ELSE
                           //PayloadLen is total Len minus topic len minus topic len info minus paket Id len
                           #statRcvMsgPayloadLen := #statRcvMsgTotalLen - #statRcvMsgTopicLen - #TWO_BYTE_LEN_INFO - #TWO_BYTE_LEN_INFO;
                         END_IF;

                         //Clear Output message:
                         #receivedTopic := #EMPTY_WSTRING;
                         //Start receiving with topic
                         #statRcvMsgDecodeState := #MSG_DECODE_STATE_TOPIC;
                         //Start Topic at first character
                         #statRcvMsgTopicPos := #FIRST_CHARACTER;
                         //Start RcvMsg at first array element
                         #statRcvMsgPayloadPos := LOWER_BOUND(ARR := #receivedMsgPayload, DIM := #ONE_DIMENSION);
                         //Set Output for received len according to array dimension
                         #tempReceivedMsgDataArrayTotalLen := ABS(UPPER_BOUND(ARR := #receivedMsgPayload, DIM := #ONE_DIMENSION) - LOWER_BOUND(ARR := #receivedMsgPayload, DIM := #ONE_DIMENSION)) + #ARRAY_LEN_OFFSET_PLUS_1;
                         IF #statRcvMsgPayloadLen < #tempReceivedMsgDataArrayTotalLen THEN
                           #statRcvMsgDataLen := #statRcvMsgPayloadLen;
                         ELSE
                           #statRcvMsgDataLen := DINT_TO_UDINT(#tempReceivedMsgDataArrayTotalLen);
                         END_IF;
                       END_REGION RECEIVED_PUBLISH_PAKET_FROM_BROKER

                     #MQTT_MSG_DECODING:
                       REGION RECEIVED_PAKET_DECODE
                         CASE #statRcvMsgDecodeState OF
                           #MSG_DECODE_STATE_NO_PROCESSING: // NO Processing
                             ;
                           #MSG_DECODE_STATE_TOPIC:  // Statement section case 1
                             #tempReceivedTopicStringMaxLen := MAX_LEN(#receivedTopic);
                             //Copy Topic To WString Inout
                             IF #statRcvMsgTopicPos <= #tempReceivedTopicStringMaxLen THEN
                               #receivedTopic[#statRcvMsgTopicPos] := BYTE_TO_WCHAR(#statRcvBuffer[#tempTrcvBufferPos]);
                               #statRcvMsgTopicPos += 1;
                             ELSE
                               //Max String len reached.
                               #statRcvMsgInternalStatus := #MSG_DECODE_STATUS_TOPIC_TOO_LONG;
                             END_IF;
                             //decrement
                             #statRcvMsgTopicLen -= 1;
                             //increment
                             #tempTrcvBufferPos += 1;
                             //Check condition, if topic fully decoded:
                             IF #statRcvMsgTopicLen <= 0 THEN
                               //Decide what to do next:
                               IF #statRcvMsgQoS > #MQTT_QOS_0 THEN
                                 //NextStep Decode PaketID
                                 #statRcvMsgDecodeState := #MSG_DECODE_STATE_PAKET_ID_MSB;
                               ELSIF #statRcvMsgQoS = #MQTT_QOS_0 AND #statRcvMsgPayloadLen > 0 THEN
                                 //NextStep Decode Payload
                                 #statRcvMsgDecodeState := #MSG_DECODE_STATE_PAYLOAD;
                               ELSE
                                 // QoS=0 and no Payload => Done
                                 // Decoding complete
                                 #statRcvMsgDecodeState := #MSG_DECODE_STATE_NO_PROCESSING;
                                 //Set New message flag
                                 IF #statRcvMsgInternalStatus = #MSG_DECODE_STATUS_NO_NEW_MSG THEN
                                   //New message received ok
                                   #statRcvMsgStatus := #MSG_DECODE_STATUS_NEW_MSG_OK;
                                 ELSE
                                   //Message received, but Payload or Topic longer than inout data area
                                   #statRcvMsgStatus := #MSG_DECODE_STATUS_TOPIC_TOO_LONG;
                                 END_IF;
                               END_IF;
                             END_IF;
                           #MSG_DECODE_STATE_PAKET_ID_MSB:  // Decode PaketId MSB
                             //Copy PaketID
                             #statRcvMsgPaketId.%B1 := #statRcvBuffer[#tempTrcvBufferPos]; //MSB
                             #tempTrcvBufferPos += 1; //Increment
                             #statRcvMsgDecodeState := #MSG_DECODE_STATE_PAKET_ID_LSB;
                           #MSG_DECODE_STATE_PAKET_ID_LSB: // Decode PaketId LSB
                             //Copy PaketID
                             #statRcvMsgPaketId.%B0 := #statRcvBuffer[#tempTrcvBufferPos]; //LSB
                             #tempTrcvBufferPos += 1; //Increment
                             IF #statRcvMsgPayloadLen > 0 THEN
                               #statRcvMsgDecodeState := #MSG_DECODE_STATE_PAYLOAD;
                             ELSE
                               // Decoding complete
                               #statRcvMsgDecodeState := #MSG_DECODE_STATE_NO_PROCESSING;
                               //Set New message flag
                               IF #statRcvMsgInternalStatus = #MSG_DECODE_STATUS_NO_NEW_MSG THEN
                                 //New message received ok
                                 #statRcvMsgStatus := #MSG_DECODE_STATUS_NEW_MSG_OK;
                               ELSE
                                 //Message received, but Payload or Topic longer than inout data area
                                 #statRcvMsgStatus := #MSG_DECODE_STATUS_TOPIC_TOO_LONG;
                               END_IF;
                               // Send PubAck Msg
                               #statSendPubAckMsg := TRUE;
                             END_IF;
                           #MSG_DECODE_STATE_PAYLOAD:
                             #tempUpperBoundRcvMsgDataArray := UPPER_BOUND(ARR := #receivedMsgPayload, DIM := #ONE_DIMENSION);

                             IF #statRcvMsgPayloadPos <= #tempUpperBoundRcvMsgDataArray THEN
                               //Copy to output
                               #receivedMsgPayload[#statRcvMsgPayloadPos] := (#statRcvBuffer[#tempTrcvBufferPos]);
                               //Increment the pos
                               #statRcvMsgPayloadPos += 1;
                             ELSE
                               //Max Payload len reached, skip
                               #statRcvMsgInternalStatus := #MSG_DECODE_STATUS_PAYLOAD_TOO_LONG;
                             END_IF;
                             //Decrement msg payload len
                             #statRcvMsgPayloadLen -= 1;
                             //Increment Buffer Pos
                             #tempTrcvBufferPos += 1;
                             //Check condition, if payload fully decoded:
                             IF #statRcvMsgPayloadLen <= 0 THEN
                               // Decoding complete
                               #statRcvMsgDecodeState := #MSG_DECODE_STATE_NO_PROCESSING;
                               //Set New message flag
                               IF #statRcvMsgInternalStatus = #MSG_DECODE_STATUS_NO_NEW_MSG THEN
                                 //New message received ok
                                 #statRcvMsgStatus := #MSG_DECODE_STATUS_NEW_MSG_OK;
                               ELSE
                                 //Message received, but Payload or Topic longer than inout data area
                                 #statRcvMsgStatus := #MSG_DECODE_STATUS_PAYLOAD_TOO_LONG;
                               END_IF;
                               //Decide if a PUB ACK needs to be send
                               IF #statRcvMsgQoS > #MQTT_QOS_0 THEN
                                 // Send PubAck Msg
                                 #statSendPubAckMsg := TRUE;
                               END_IF;
                             END_IF;
                           ELSE
                             //else case
                             #statStatus := #ERR_UNDEFINED_STATE;
                             #statErrorUserCleared := TRUE;
                             ;
                         END_CASE;
                       END_REGION RECEIVED_PAKET_DECODE
                     ELSE // No Header found, SKIP entry of buffer:
                       #tempTrcvBufferPos += 1;
                   END_CASE;
                 END_WHILE;
               END_REGION TRCV_NEW_DATA
             END_IF;

